modbus_var[0] :=%IW0;
Temp_chilled_medium_out:=wordstoReal(modbus_var_1000[0],modbus_var_1000[1]);
Temp_chilled_medium_in:=wordstoReal(modbus_var_1000[2],modbus_var_1000[3]);
Temp_water_inlet_cond:=wordstoReal(modbus_var_1000[4],modbus_var_1000[5]);
Temp_water_outlet_cond:=wordstoReal(modbus_var_1000[6],modbus_var_1000[7]);
SP_CW_controller:=wordstoReal(modbus_var_1000[8],modbus_var_1000[9]);
SP_PID_seawater:=wordstoReal(modbus_var_1000[10],modbus_var_1000[11]);
COP_chiller_mech:=wordstoReal(modbus_var_1000[12],modbus_var_1000[13]);
P2_mot_1_kW:=wordstoReal(modbus_var_1000[14],modbus_var_1000[15]);
Thrust_bearing_ref:=wordstoReal(modbus_var_1000[16],modbus_var_1000[17]);
Thrust_bearing_ref_min:=wordstoReal(modbus_var_1000[18],modbus_var_1000[19]);
Thrust_bearing_ref_max:=wordstoReal(modbus_var_1000[20],modbus_var_1000[21]);
Press_suction_compr:=wordstoReal(modbus_var_1000[22],modbus_var_1000[23]);
Press_discharge_compr:=wordstoReal(modbus_var_1000[24],modbus_var_1000[25]);
Suction_saturated_temp:=wordstoReal(modbus_var_1000[26],modbus_var_1000[27]);
Discharge_saturated_temp:=wordstoReal(modbus_var_1000[28],modbus_var_1000[29]);
Temp_discharge:=wordstoReal(modbus_var_1000[30],modbus_var_1000[31]);
Discharge_superheat:=wordstoReal(modbus_var_1000[32],modbus_var_1000[33]);
Liquid_level_condenser:=wordstoReal(modbus_var_1000[34],modbus_var_1000[35]);
Feedback_liquid_valve:=wordstoReal(modbus_var_1000[36],modbus_var_1000[37]);
Feedback_HGV:=wordstoReal(modbus_var_1000[38],modbus_var_1000[39]);
Spare_0:=wordstoReal(modbus_var_1000[40],modbus_var_1000[41]);
Chiller_capacity_kW:=wordstoReal(modbus_var_1000[42],modbus_var_1000[43]);
Motor_current:=wordstoReal(modbus_var_1000[44],modbus_var_1000[45]);
SP_MC_controller:=wordstoReal(modbus_var_1000[46],modbus_var_1000[47]);
Running_hours_compressormotor:=wordstoReal(modbus_var_1000[48],modbus_var_1000[49]);   //wordstoReal yes
//Running_hours_compressormotor:=wordstoDword(modbus_var_1000[48],modbus_var_1000[49]);     //wordstoDword nope
Chiller_capacity_t1:=wordstoReal(modbus_var_1000[50],modbus_var_1000[51]);
Thrust_bearing_position:=wordstoReal(modbus_var_1000[52],modbus_var_1000[53]);
Feedback_PRV:=wordstoReal(modbus_var_1000[54],modbus_var_1000[55]);
Prerotary_output:=wordstoReal(modbus_var_1000[56],modbus_var_1000[57]);
Feedback_VGD:=wordstoReal(modbus_var_1000[58],modbus_var_1000[59]);
VGD_output:=wordstoReal(modbus_var_1000[60],modbus_var_1000[61]);
Hot_gas_valve_output:=wordstoReal(modbus_var_1000[62],modbus_var_1000[63]);
Anti_recycle_time:=wordstoReal(modbus_var_1000[64],modbus_var_1000[65]);
Spare:=wordstoReal(modbus_var_1000[66],modbus_var_1000[67]);
Speed_feedback_VFD:=wordstoReal(modbus_var_1000[68],modbus_var_1000[69]);
Spare:=wordstoReal(modbus_var_1000[70],modbus_var_1000[71]);
Stall_detector:=wordstoReal(modbus_var_1000[72],modbus_var_1000[73]);
Chiller_capacity:=wordstoReal(modbus_var_1000[74],modbus_var_1000[75]);
Spare:=wordstoReal(modbus_var_1000[76],modbus_var_1000[77]);
Spare:=wordstoReal(modbus_var_1000[78],modbus_var_1000[79]);
Press_oil_receiver:=wordstoReal(modbus_var_1000[80],modbus_var_1000[81]);
Press_oil_compr:=wordstoReal(modbus_var_1000[82],modbus_var_1000[83]);
Oil_pressure_before_filter:=wordstoReal(modbus_var_1000[84],modbus_var_1000[85]);
Oil_diff_pressure:=wordstoReal(modbus_var_1000[86],modbus_var_1000[87]);
SP_freq_oil_pump_VFD:=wordstoReal(modbus_var_1000[88],modbus_var_1000[89]); 
//Setpoint_conv_oil_pump:=wordstoReal(modbus_var_1000[88],modbus_var_1000[89]); 
Oil_temp_receiver:=wordstoReal(modbus_var_1000[90],modbus_var_1000[91]);
Temp_oil_inlet_compr:=wordstoReal(modbus_var_1000[92],modbus_var_1000[93]);
SP_oil_pressure_diff:=wordstoReal(modbus_var_1000[94],modbus_var_1000[95]);
Oil_pump_running_hours:=wordstoReal(modbus_var_1000[96],modbus_var_1000[97]);
Spare:=wordstoReal(modbus_var_1000[98],modbus_var_1000[99]);
Spare:=wordstoReal(modbus_var_1000[100],modbus_var_1000[101]);
Spare:=wordstoReal(modbus_var_1000[102],modbus_var_1000[103]);
Press_chilled_medium_out:=wordstoReal(modbus_var_1000[104],modbus_var_1000[105]);
Press_chilled_medium_in:=wordstoReal(modbus_var_1000[106],modbus_var_1000[107]);
Press_water_cond_out:=wordstoReal(modbus_var_1000[108],modbus_var_1000[109]);
Press_water_cond_inlet:=wordstoReal(modbus_var_1000[110],modbus_var_1000[111]);
dP_CW:=wordstoReal(modbus_var_1000[112],modbus_var_1000[113]);
dP_SW:=wordstoReal(modbus_var_1000[114],modbus_var_1000[115]);
Feedback_seawater_valve_overboard:=wordstoReal(modbus_var_1000[116],modbus_var_1000[117]);
Spare:=wordstoReal(modbus_var_1000[118],modbus_var_1000[119]);
Spare:=wordstoReal(modbus_var_1000[120],modbus_var_1000[121]);
Spare:=wordstoReal(modbus_var_1000[122],modbus_var_1000[123]);
Temp_motor_wind_R:=wordstoReal(modbus_var_1001[124],modbus_var_1001[125]);
Temp_motor_wind_S:=wordstoReal(modbus_var_1001[126],modbus_var_1001[127]);
Temp_motor_wind_T:=wordstoReal(modbus_var_1001[128],modbus_var_1001[129]);
Max_motor_wind_temp:=wordstoReal(modbus_var_1001[130],modbus_var_1001[131]);
Temp_motor_air:=wordstoReal(modbus_var_1001[132],modbus_var_1001[133]);
Temp_motor_bearing_DE:=wordstoReal(modbus_var_1001[134],modbus_var_1001[135]);
Temp_motor_bearing_NDE:=wordstoReal(modbus_var_1001[136],modbus_var_1001[137]);
Vibration_compressor_DE:=wordstoReal(modbus_var_1001[138],modbus_var_1001[139]);
Vibration_compressor_NDE:=wordstoReal(modbus_var_1001[140],modbus_var_1001[141]);
SW_pump_speed_order:=wordstoReal(modbus_var_1001[142],modbus_var_1001[143]);
Order_SWW_overboard:=wordstoReal(modbus_var_1001[144],modbus_var_1001[145]);
Control_signal_SW_valve:=wordstoReal(modbus_var_1001[144],modbus_var_1001[145]);   
Order_SWW_bypass:=wordstoReal(modbus_var_1001[146],modbus_var_1001[147]);
Liquid_valve_output:=wordstoReal(modbus_var_1001[148],modbus_var_1001[149]);
SP_cond_press:=wordstoReal(modbus_var_1001[150],modbus_var_1001[151]);
SP_PID_Level:=wordstoReal(modbus_var_1001[152],modbus_var_1001[153]);  //mer rätt AO?
//SP_t1:=wordstoReal(modbus_var_1001[152],modbus_var_1001[153]);       // vad är detta måste kollas  SP Condenser level? PT   Tror Discharge pressure setpoint AÖ
Oil_Filter_Drop:=wordstoReal(modbus_var_1001[154],modbus_var_1001[155]);    
Min_allowed_PRVposition:=wordstoReal(modbus_var_1001[156],modbus_var_1001[157]); 
Stall_ramp:=wordstoReal(modbus_var_1001[158],modbus_var_1001[159]);
Theta_out:=wordstoReal(modbus_var_1001[160],modbus_var_1001[161]);
Control_signal_unit_d:=wordstoReal(modbus_var_1001[162],modbus_var_1001[163]);    // Sequence control signal  PT
Order_VFD_perc:=wordstoReal(modbus_var_1001[164],modbus_var_1001[165]); 
Order_VFD_Hz:=wordstoReal(modbus_var_1001[166],modbus_var_1001[167]);
Speed_feedback_VFD:=wordstoReal(modbus_var_1001[168],modbus_var_1001[169]);
Opt_speed_VFD_perc:=wordstoReal(modbus_var_1001[170],modbus_var_1001[171]);
Opt_speed_VFD_Hz:=wordstoReal(modbus_var_1001[172],modbus_var_1001[173]);
Spare:=wordstoReal(modbus_var_1001[174],modbus_var_1001[175]);
P1_motor_kW:=wordstoReal(modbus_var_1001[176],modbus_var_1001[177]);
COP_chiller_ele:=wordstoReal(modbus_var_1001[178],modbus_var_1001[179]);
PI_chiller:=wordstoReal(modbus_var_1001[180],modbus_var_1001[181]);
Wasted_energy_kW:=wordstoReal(modbus_var_1001[182],modbus_var_1001[183]);
Cal_date_MMYY:=wordstoReal(modbus_var_1001[184],modbus_var_1001[185]);
Spare:=wordstoReal(modbus_var_1001[186],modbus_var_1001[187]);
Spare:=wordstoReal(modbus_var_1001[188],modbus_var_1001[189]);
Spare:=wordstoReal(modbus_var_1001[190],modbus_var_1001[191]);
Spare:=wordstoReal(modbus_var_1001[192],modbus_var_1001[193]);
Spare:=wordstoReal(modbus_var_1001[194],modbus_var_1001[195]);
Spare:=wordstoReal(modbus_var_1001[196],modbus_var_1001[197]);
Spare:=wordstoReal(modbus_var_1001[198],modbus_var_1001[199]);
Spare:=wordstoReal(modbus_var_1001[200],modbus_var_1001[201]);
Spare:=wordstoReal(modbus_var_1001[202],modbus_var_1001[203]);
Spare:=wordstoReal(modbus_var_1001[204],modbus_var_1001[205]);
Spare:=wordstoReal(modbus_var_1001[206],modbus_var_1001[207]);
Spare:=wordstoReal(modbus_var_1001[208],modbus_var_1001[209]);
Spare:=wordstoReal(modbus_var_1001[210],modbus_var_1001[211]);

// Write PI to PLC
modbus_var_1001[180]:=modbusslave_com.sequence_highByte_PI_ch_1;
modbus_var_1001[181]:=modbusslave_com.sequence_lowByte_PI_ch_1;
modbus_var_1001[182]:=modbusslave_com.sequence_highByte_Wasted_energy_ch_1_kW;
modbus_var_1001[183]:=modbusslave_com.sequence_lowByte_Wasted_energy_ch_1_kW;

// Word variables
Alarm_limit_stall_count_unscaled:=modbus_var_1001[211];
Alarm_limit_stall_count:=Alarm_limit_stall_count_unscaled*1.0;
Sec_above_stall_limit:=scaleFunction(modbus_var_1001[212],1.0, 0);
Min_above_stall_limit:=scaleFunction(modbus_var_1001[213],1.0, 0);
Hrs_above_stall_limit:=scaleFunction(modbus_var_1001[214],1.0, 0);
Days_above_stall_limit:=scaleFunction(modbus_var_1001[215],1.0, 0);
Number_of_starts:=scaleFunction(modbus_var_1001[216],1.0, 0);
Q2_chillerMWh:=scaleFunction(modbus_var_1001[217],1.0, 0); 
Chiller_P2_MWh:=scaleFunction(modbus_var_1001[218],1.0, 0);
Surge_counter_VFD:=scaleFunction(modbus_var_1001[219],1.0, 0);

Trip_BITs_0_to_15:=modbus_var_1002[320];
Trip_BITs_16_to_31:=modbus_var_1002[321];
Trip_BITs_32_to_47:=modbus_var_1002[322];
Trip_BITs_48_to_63:=modbus_var_1002[323];
Trip_BITs_64_to_79:=modbus_var_1002[324];
Trip_BITs_80_to_95:=modbus_var_1002[325];
Trip_BITs_96_to_121:=modbus_var_1002[326];
Trip_BITs_122_to_137:=modbus_var_1002[327];
Trip_BITs_138_to_153:=modbus_var_1002[328];

Alarm_BITs_0_to_15:=modbus_var_1002[330];
Alarm_BITs_16_to_31:=modbus_var_1002[331];
Alarm_BITs_32_to_47:=modbus_var_1002[332];
Alarm_BITs_48_to_63:=modbus_var_1002[332];
Alarm_BITs_64_to_79:=modbus_var_1002[333];

Statusbits_0_to_15:=modbus_var_1002[300];
Statusbits_16_to_31:=modbus_var_1002[301];
Statusbits_32_to_47:=modbus_var_1002[302];
Statusbits_48_to_63:=modbus_var_1002[303];
Statusbits_64_to_79:=modbus_var_1002[304];
Statusbits_80_to_95:=modbus_var_1002[305];
Statusbits_96_to_111:=modbus_var_1002[310];
Statusbits_112_to_127:=modbus_var_1002[311];


//320
T_Overload_compressor_motor:=maskbitFunction(Trip_BITs_0_to_15,0);
T_Starter_failure_trip:=maskbitFunction(Trip_BITs_0_to_15,1);
T_Oil_pump_running_failure:=maskbitFunction(Trip_BITs_0_to_15,2);
T_Overload_oil_pump_motor:=maskbitFunction(Trip_BITs_0_to_15,3);
T_Compressor_running_failure:=maskbitFunction(Trip_BITs_0_to_15,4);
T_Softstarter_failure:=maskbitFunction(Trip_BITs_0_to_15,5);
T_Motorstarter_failure:=maskbitFunction(Trip_BITs_0_to_15,6);
T_Comp_motor_power_loss:=maskbitFunction(Trip_BITs_0_to_15,7);
T_Emergency_stop:=maskbitFunction(Trip_BITs_0_to_15,8);
T_Flow_switch_FT01:=maskbitFunction(Trip_BITs_0_to_15,9);
T_Chilled_pump_run_failure:=maskbitFunction(Trip_BITs_0_to_15,10);
T_CW_valveopen_failure:=maskbitFunction(Trip_BITs_0_to_15,11);
T_Sea_water_pump_run_failure:=maskbitFunction(Trip_BITs_0_to_15,12);
T_SW_valveopen_failure:=maskbitFunction(Trip_BITs_0_to_15,13);
T_Comp_motor_leak_detection:=maskbitFunction(Trip_BITs_0_to_15,14);
T_Cathodic_protect_sys_alarm:=maskbitFunction(Trip_BITs_0_to_15,15);
//321
T_High_discharge_pressure:=maskbitFunction(Trip_BITs_16_to_31,0);
T_Low_discharge_pressure:=maskbitFunction(Trip_BITs_16_to_31,1);
T_Low_suction_pressure:=maskbitFunction(Trip_BITs_16_to_31,2);
T_High_suction_pressure:=maskbitFunction(Trip_BITs_16_to_31,3);
T_High_discharge_temp:=maskbitFunction(Trip_BITs_16_to_31,4);
T_High_temp_oil_inlet_comp:=maskbitFunction(Trip_BITs_16_to_31,5);
T_High_temp_oil_receiver:=maskbitFunction(Trip_BITs_16_to_31,6);
T_Low_temp_oil_receiver:=maskbitFunction(Trip_BITs_16_to_31,7);
T_Low_oil_diff_pressure:=maskbitFunction(Trip_BITs_16_to_31,8);
T_High_diff_oil_pressure:=maskbitFunction(Trip_BITs_16_to_31,9);
T_High_oil_filter_diff_press:=maskbitFunction(Trip_BITs_16_to_31,10);
T_High_disch_superheat:=maskbitFunction(Trip_BITs_16_to_31,11);
T_Low_disch_superheat:=maskbitFunction(Trip_BITs_16_to_31,12);
T_Low_CW_inlet_temp:=maskbitFunction(Trip_BITs_16_to_31,13);
T_High_CW_inlet_temp:=maskbitFunction(Trip_BITs_16_to_31,14);
T_Low_CW_outlet_temp:=maskbitFunction(Trip_BITs_16_to_31,15);
//322
T_High_CW_outlet_temp:=maskbitFunction(Trip_BITs_32_to_47,0);
T_Low_chilled_medium_flow:=maskbitFunction(Trip_BITs_32_to_47,1);
T_High_chilled_medium_flow:=maskbitFunction(Trip_BITs_32_to_47,2);
T_Low_SW_inlet_temp:=maskbitFunction(Trip_BITs_32_to_47,3);
T_High_SW_inlet_temp:=maskbitFunction(Trip_BITs_32_to_47,4);
T_Low_SW_outlet_temp:=maskbitFunction(Trip_BITs_32_to_47,5);
T_High_SW_outlet_temp:=maskbitFunction(Trip_BITs_32_to_47,6);
T_Low_condenser_flow:=maskbitFunction(Trip_BITs_32_to_47,7);
T_High_condenser_flow:=maskbitFunction(Trip_BITs_32_to_47,8);
T_High_motor_wind_temp_R:=maskbitFunction(Trip_BITs_32_to_47,9);
T_High_motor_wind_temp_S:=maskbitFunction(Trip_BITs_32_to_47,10);
T_High_motor_wind_temp_T:=maskbitFunction(Trip_BITs_32_to_47,11);
T_High_comp_mot_DE_bear_temp:=maskbitFunction(Trip_BITs_32_to_47,12);
T_High_comp_mot_NDE_bear_temp:=maskbitFunction(Trip_BITs_32_to_47,13);
T_High_motor_air_temp:=maskbitFunction(Trip_BITs_32_to_47,14);
T_High_comp_mot_DE_bear_vib:=maskbitFunction(Trip_BITs_32_to_47,15);
//323
T_High_comp_mot_NDE_bear_vib:=maskbitFunction(Trip_BITs_48_to_63,0);
T_High_press_ratio:=maskbitFunction(Trip_BITs_48_to_63,1);
T_Low_press_ratio:=maskbitFunction(Trip_BITs_48_to_63,2);
T_High_CW_dP:=maskbitFunction(Trip_BITs_48_to_63,3);
T_Low_CW_dP:=maskbitFunction(Trip_BITs_48_to_63,4);
T_High_SW_dP:=maskbitFunction(Trip_BITs_48_to_63,5);
T_Low_SW_dP:=maskbitFunction(Trip_BITs_48_to_63,6);
T_Long_time_PRV:=maskbitFunction(Trip_BITs_48_to_63,7);
T_Surge_detection:=maskbitFunction(Trip_BITs_48_to_63,8);
T_Comp_thrust_bearing_position:=maskbitFunction(Trip_BITs_48_to_63,9);
T_Comp_thrust_neg_move:=maskbitFunction(Trip_BITs_48_to_63,10);
T_Comp_thrust_pos_move:=maskbitFunction(Trip_BITs_48_to_63,11);
T_VGD_fault:=maskbitFunction(Trip_BITs_48_to_63,12);
T_Low_liquid_level:=maskbitFunction(Trip_BITs_48_to_63,13);
T_Low_oilpress_prelube:=maskbitFunction(Trip_BITs_48_to_63,14);
T_Low_oilpress_standby:=maskbitFunction(Trip_BITs_48_to_63,15);
//324
T_Sensor_low_signal_AI_64 :=maskbitFunction(Trip_BITs_64_to_79,0);
T_Sensor_high_signal_AI_64 :=maskbitFunction(Trip_BITs_64_to_79,1);
T_Sensor_low_signal_AI_66 :=maskbitFunction(Trip_BITs_64_to_79,2);
T_Sensor_high_signal_AI_66 :=maskbitFunction(Trip_BITs_64_to_79,3);
T_Sensor_low_signal_AI_128 :=maskbitFunction(Trip_BITs_64_to_79,4);
T_Sensor_high_signal_AI_128 :=maskbitFunction(Trip_BITs_64_to_79,5);
T_Sensor_low_signal_AI_130 :=maskbitFunction(Trip_BITs_64_to_79,6);
T_Sensor_high_signal_AI_130 :=maskbitFunction(Trip_BITs_64_to_79,7);
T_Sensor_low_signal_AI_132 :=maskbitFunction(Trip_BITs_64_to_79,8);
T_Sensor_high_signal_AI_132 :=maskbitFunction(Trip_BITs_64_to_79,9);
T_Sensor_low_signal_AI_134 :=maskbitFunction(Trip_BITs_64_to_79,10);
T_Sensor_high_signal_AI_134 :=maskbitFunction(Trip_BITs_64_to_79,11);
T_Sensor_low_signal_AI_136 :=maskbitFunction(Trip_BITs_64_to_79,12);
T_Sensor_high_signal_AI_136 :=maskbitFunction(Trip_BITs_64_to_79,13);
T_Sensor_low_signal_AI_138 :=maskbitFunction(Trip_BITs_64_to_79,14);
T_Sensor_high_signal_AI_138 :=maskbitFunction(Trip_BITs_64_to_79,15);

T_Sensor_low_signal_AI_140 :=maskbitFunction(Trip_BITs_80_to_95,0);
T_Sensor_high_signal_AI_140 :=maskbitFunction(Trip_BITs_80_to_95,1);
T_Sensor_low_signal_AI_142 :=maskbitFunction(Trip_BITs_80_to_95,2);
T_Sensor_high_signal_AI_142 :=maskbitFunction(Trip_BITs_80_to_95,3);
T_Sensor_low_signal_AI_144 :=maskbitFunction(Trip_BITs_80_to_95,4);
T_Sensor_high_signal_AI_144 :=maskbitFunction(Trip_BITs_80_to_95,5);
T_Sensor_low_signal_AI_146 :=maskbitFunction(Trip_BITs_80_to_95,6);
T_Sensor_high_signal_AI_146 :=maskbitFunction(Trip_BITs_80_to_95,7);
T_Sensor_low_signal_AI_148 :=maskbitFunction(Trip_BITs_80_to_95,8);
T_Sensor_high_signal_AI_148 :=maskbitFunction(Trip_BITs_80_to_95,9);
T_Sensor_low_signal_AI_150 :=maskbitFunction(Trip_BITs_80_to_95,10);
T_Sensor_high_signal_AI_150 :=maskbitFunction(Trip_BITs_80_to_95,11);
T_Sensor_low_signal_AI_152 :=maskbitFunction(Trip_BITs_80_to_95,12);
T_Sensor_high_signal_AI_152 :=maskbitFunction(Trip_BITs_80_to_95,13);
T_Sensor_low_signal_AI_154 :=maskbitFunction(Trip_BITs_80_to_95,14);
T_Sensor_high_signal_AI_154 :=maskbitFunction(Trip_BITs_80_to_95,15);

T_Sensor_low_signal_AI_156 :=maskbitFunction(Trip_BITs_96_to_121,0);
T_Sensor_high_signal_AI_156 :=maskbitFunction(Trip_BITs_96_to_121,1);
T_Sensor_low_signal_AI_158 :=maskbitFunction(Trip_BITs_96_to_121,2);
T_Sensor_high_signal_AI_158 :=maskbitFunction(Trip_BITs_96_to_121,3);
T_Sensor_low_signal_AI_160 :=maskbitFunction(Trip_BITs_96_to_121,4);
T_Sensor_high_signal_AI_160 :=maskbitFunction(Trip_BITs_96_to_121,5);
T_Sensor_low_signal_AI_162 :=maskbitFunction(Trip_BITs_96_to_121,6);
T_Sensor_high_signal_AI_162 :=maskbitFunction(Trip_BITs_96_to_121,7);
T_Sensor_low_signal_AI_164 :=maskbitFunction(Trip_BITs_96_to_121,8);
T_Sensor_high_signal_AI_164 :=maskbitFunction(Trip_BITs_96_to_121,9);
T_Sensor_low_signal_AI_166 :=maskbitFunction(Trip_BITs_96_to_121,10);
T_Sensor_high_signal_AI_166 :=maskbitFunction(Trip_BITs_96_to_121,11);
T_Sensor_low_signal_AI_168 :=maskbitFunction(Trip_BITs_96_to_121,12);
T_Sensor_high_signal_AI_168 :=maskbitFunction(Trip_BITs_96_to_121,13);
T_Sensor_low_signal_AI_170 :=maskbitFunction(Trip_BITs_96_to_121,14);
T_Sensor_high_signal_AI_170 :=maskbitFunction(Trip_BITs_96_to_121,15);

T_Sensor_low_signal_AI_172 :=maskbitFunction(Trip_BITs_122_to_137,0);
T_Sensor_high_signal_AI_172 :=maskbitFunction(Trip_BITs_122_to_137,1);
T_Sensor_low_signal_AI_174 :=maskbitFunction(Trip_BITs_122_to_137,2);
T_Sensor_high_signal_AI_174 :=maskbitFunction(Trip_BITs_122_to_137,3);
T_Sensor_high_signal_AI_176 :=maskbitFunction(Trip_BITs_122_to_137,4);
T_Sensor_high_signal_AI_178 :=maskbitFunction(Trip_BITs_122_to_137,5);
T_Sensor_high_signal_AI_180 :=maskbitFunction(Trip_BITs_122_to_137,6);
T_Sensor_high_signal_AI_182 :=maskbitFunction(Trip_BITs_122_to_137,7);
T_Sensor_high_signal_AI_184 :=maskbitFunction(Trip_BITs_122_to_137,8);
T_Sensor_high_signal_AI_186 :=maskbitFunction(Trip_BITs_122_to_137,9);
T_Sensor_high_signal_AI_188 :=maskbitFunction(Trip_BITs_122_to_137,10);
T_Sensor_high_signal_AI_190 :=maskbitFunction(Trip_BITs_122_to_137,11);
T_Sensor_high_signal_AI_192 :=maskbitFunction(Trip_BITs_122_to_137,12);
T_Sensor_high_signal_AI_194 :=maskbitFunction(Trip_BITs_122_to_137,13);
T_Sensor_high_signal_AI_196 :=maskbitFunction(Trip_BITs_122_to_137,14);
T_Sensor_high_signal_AI_198 :=maskbitFunction(Trip_BITs_122_to_137,15);

T_Sensor_high_signal_AI_200 :=maskbitFunction(Trip_BITs_138_to_153,0);
T_Sensor_high_signal_AI_202 :=maskbitFunction(Trip_BITs_138_to_153,1);
T_Sensor_high_signal_AI_204 :=maskbitFunction(Trip_BITs_138_to_153,2);
T_Sensor_high_signal_AI_206:=maskbitFunction(Trip_BITs_138_to_153,3);

// Alarm bits 330
A_High_control_panel_temp:=maskbitFunction(Alarm_BITs_0_to_15,0);
A_high_disch_press:=maskbitFunction(Alarm_BITs_0_to_15,1);
A_low_disch_press :=maskbitFunction(Alarm_BITs_0_to_15,2);
A_Low_suction_pressure:=maskbitFunction(Alarm_BITs_0_to_15,3);
A_High_suction_pressure:=maskbitFunction(Alarm_BITs_0_to_15,4);
A_High_discharge_temp :=maskbitFunction(Alarm_BITs_0_to_15,5);
A_High_temp_oil_inlet_comp:=maskbitFunction(Alarm_BITs_0_to_15,6);
A_Low_temp_oil_inlet_comp:=maskbitFunction(Alarm_BITs_0_to_15,7);
A_High_oil_temp_receiver:=maskbitFunction(Alarm_BITs_0_to_15,8);
A_Low_oil_temp_receiver:=maskbitFunction(Alarm_BITs_0_to_15,9);
A_Low_oil_diff_pressure:=maskbitFunction(Alarm_BITs_0_to_15,10);
A_High_oil_diff_pressure:=maskbitFunction(Alarm_BITs_0_to_15,11);
A_High_discharge_superheat:=maskbitFunction(Alarm_BITs_0_to_15,12);
A_Low_discharge_superheat:=maskbitFunction(Alarm_BITs_0_to_15,13);
A_Low_CW_inlet_temp:=maskbitFunction(Alarm_BITs_0_to_15,14);
A_High_CW_inlet_temp:=maskbitFunction(Alarm_BITs_0_to_15,15);
//331
A_Low_CW_outlet_temp:=maskbitFunction(Alarm_BITs_16_to_31,0);
A_High_CW_outlet_temp:=maskbitFunction(Alarm_BITs_16_to_31,1);
A_Low_chilled_medium_flow:=maskbitFunction(Alarm_BITs_16_to_31,2);
A_High_chilled_medium_flow:=maskbitFunction(Alarm_BITs_16_to_31,3);
A_Low_condenser_flow:=maskbitFunction(Alarm_BITs_16_to_31,4);
A_High_condenser_flow:=maskbitFunction(Alarm_BITs_16_to_31,5);
A_High_press_ratio:=maskbitFunction(Alarm_BITs_16_to_31,6);
A_Low_press_ratio:=maskbitFunction(Alarm_BITs_16_to_31,7);
A_Motor_speed_low :=maskbitFunction(Alarm_BITs_16_to_31,8);
A_Low_SW_inlet_temp:=maskbitFunction(Alarm_BITs_16_to_31,9); 
A_High_SW_inlet_temp:=maskbitFunction(Alarm_BITs_16_to_31,10); 
A_Low_SW_outlet_temp:=maskbitFunction(Alarm_BITs_16_to_31,11); 
A_High_SW_outlet_temp:=maskbitFunction(Alarm_BITs_16_to_31,12);
A_High_suction_superheat:=maskbitFunction(Alarm_BITs_16_to_31,13);
A_Low_suction_superheat:=maskbitFunction(Alarm_BITs_16_to_31,14);
A_High_oil_filter_diff_press:=maskbitFunction(Alarm_BITs_16_to_31,15);
//332
A_High_CW_dP:=maskbitFunction(Alarm_BITs_32_to_47,0);
A_Low_CW_dP:=maskbitFunction(Alarm_BITs_32_to_47,1);
A_High_temp_oil_separator:=maskbitFunction(Alarm_BITs_32_to_47,2);
A_Low_temp_oil_separator:=maskbitFunction(Alarm_BITs_32_to_47,3);
A_High_motor_wind_temp_R:=maskbitFunction(Alarm_BITs_32_to_47,4);
A_High_motor_wind_temp_S:=maskbitFunction(Alarm_BITs_32_to_47,5);
A_High_motor_wind_temp_T:=maskbitFunction(Alarm_BITs_32_to_47,6);
A_High_comp_mo_DE_bear_temp:=maskbitFunction(Alarm_BITs_32_to_47,7);
A_High_comp_mo_NDE_bear_temp:=maskbitFunction(Alarm_BITs_32_to_47,8);
A_High_motor_air_temp:=maskbitFunction(Alarm_BITs_32_to_47,9);
A_High_comp_mo_DE_bear_vib:=maskbitFunction(Alarm_BITs_32_to_47,10);
A_High_comp_mo_NDE_bear_vib:=maskbitFunction(Alarm_BITs_32_to_47,11);
//A_High_CW_dP:=maskbitFunction(Alarm_BITs_32_to_47,12);                       //Double defined?
//A_Low_CW_dP:=maskbitFunction(Alarm_BITs_32_to_47,13);                        //Double defined?
A_High_SW_dP:=maskbitFunction(Alarm_BITs_32_to_47,14);                       
A_Low_SW_dP:=maskbitFunction(Alarm_BITs_32_to_47,15);
//333
A_VGD_fault:=maskbitFunction(Alarm_BITs_48_to_63,0);
//A_Rotating_stall:=maskbitFunction(Alarm_BITs_48_to_63,0);  // kollas
A_Low_liquid_level:=maskbitFunction(Alarm_BITs_48_to_63,1);





// Statusbits 310
Unit_running:=maskbitFunction(Statusbits_96_to_111,0);
Unit_trip:=maskbitFunction(Statusbits_96_to_111,1);
Unit_alarm:=maskbitFunction(Statusbits_96_to_111,2);
Unit_remote:=maskbitFunction(Statusbits_96_to_111,3);
Unit_auto:=maskbitFunction(Statusbits_96_to_111,4);
Unit_manual:=maskbitFunction(Statusbits_96_to_111,5);
Unit_available:=maskbitFunction(Statusbits_96_to_111,6);
Unit_start_switch:=maskbitFunction(Statusbits_96_to_111,7);
Comp_oil_pump:=maskbitFunction(Statusbits_96_to_111,8);
Oil_heater:=maskbitFunction(Statusbits_96_to_111,9);
Solenoid_oil_return:=maskbitFunction(Statusbits_96_to_111,10);
Solenoid_liquid_inj:=maskbitFunction(Statusbits_96_to_111,11);
Low_oil_temperature:=maskbitFunction(Statusbits_96_to_111,12);
Sea_water_pump:=maskbitFunction(Statusbits_96_to_111,13);
CW_Flow_ind:=maskbitFunction(Statusbits_96_to_111,14);
Start_inhib_time_between_start:=maskbitFunction(Statusbits_96_to_111,15);
// Statusbits 311
Start_inhib_time_beetween_stop:=maskbitFunction(Statusbits_112_to_127,0);
Start_inhib_PRV_not_min:=maskbitFunction(Statusbits_112_to_127,1);
Start_inhib_Motor_overload:=maskbitFunction(Statusbits_112_to_127,2);
VFD_ready:=maskbitFunction(Statusbits_112_to_127,3);
VFD_ramp_100_perc:=maskbitFunction(Statusbits_112_to_127,4);
VFD_locked_100_perc:=maskbitFunction(Statusbits_112_to_127,5);
VFD_ramp_d_PRVcontrol:=maskbitFunction(Statusbits_112_to_127,6);
PRV_control:=maskbitFunction(Statusbits_112_to_127,7);
VFD_control:=maskbitFunction(Statusbits_112_to_127,8);
S_Spare_1:=maskbitFunction(Statusbits_112_to_127,9);
S_Spare_1:=maskbitFunction(Statusbits_112_to_127,10);
S_Spare_1:=maskbitFunction(Statusbits_112_to_127,11);
S_Spare_1:=maskbitFunction(Statusbits_112_to_127,12);
S_Spare_1:=maskbitFunction(Statusbits_112_to_127,13);
S_Spare_1:=maskbitFunction(Statusbits_112_to_127,14);
S_Spare_1:=maskbitFunction(Statusbits_112_to_127,15);

DI_0_0:=maskbitFunction(Statusbits_0_to_15,0);
DI_0_1:=maskbitFunction(Statusbits_0_to_15,1);
DI_0_2:=maskbitFunction(Statusbits_0_to_15,2);
DI_0_3:=maskbitFunction(Statusbits_0_to_15,3);
DI_0_4:=maskbitFunction(Statusbits_0_to_15,4);
DI_0_5:=maskbitFunction(Statusbits_0_to_15,5);
DI_0_6:=maskbitFunction(Statusbits_0_to_15,6);
DI_0_7:=maskbitFunction(Statusbits_0_to_15,7);
DI_1_0:=maskbitFunction(Statusbits_0_to_15,8);
DI_1_1:=maskbitFunction(Statusbits_0_to_15,9);
DI_1_2:=maskbitFunction(Statusbits_0_to_15,10);
DI_1_3:=maskbitFunction(Statusbits_0_to_15,11);
DI_1_4:=maskbitFunction(Statusbits_0_to_15,12);
DI_1_5:=maskbitFunction(Statusbits_0_to_15,13);
DI_8_0:=maskbitFunction(Statusbits_0_to_15,14);
DI_8_1:=maskbitFunction(Statusbits_0_to_15,15);

DI_8_2:=maskbitFunction(Statusbits_16_to_31,0);
DI_8_3:=maskbitFunction(Statusbits_16_to_31,1);
DI_8_4:=maskbitFunction(Statusbits_16_to_31,2);
DI_8_5:=maskbitFunction(Statusbits_16_to_31,3);
DI_8_6:=maskbitFunction(Statusbits_16_to_31,4);
DI_8_7:=maskbitFunction(Statusbits_16_to_31,5);
DI_9_0:=maskbitFunction(Statusbits_16_to_31,6);
DI_9_1:=maskbitFunction(Statusbits_16_to_31,7);
DI_9_2:=maskbitFunction(Statusbits_16_to_31,8);
DI_9_3:=maskbitFunction(Statusbits_16_to_31,9);
DI_9_4:=maskbitFunction(Statusbits_16_to_31,10);
DI_9_5:=maskbitFunction(Statusbits_16_to_31,11);
DI_9_6:=maskbitFunction(Statusbits_16_to_31,12);
DI_9_7:=maskbitFunction(Statusbits_16_to_31,13);
T_Spare_3:=maskbitFunction(Statusbits_16_to_31,14);
T_Spare_3:=maskbitFunction(Statusbits_16_to_31,15);

DO_0_0:=maskbitFunction(Statusbits_32_to_47,0);
DO_0_1:=maskbitFunction(Statusbits_32_to_47,1);
DO_0_2:=maskbitFunction(Statusbits_32_to_47,2);
DO_0_3:=maskbitFunction(Statusbits_32_to_47,3);
DO_0_4:=maskbitFunction(Statusbits_32_to_47,4);
DO_0_5:=maskbitFunction(Statusbits_32_to_47,5);
DO_0_6:=maskbitFunction(Statusbits_32_to_47,6);
DO_0_7:=maskbitFunction(Statusbits_32_to_47,7);
DO_1_0:=maskbitFunction(Statusbits_32_to_47,8);
DO_1_1:=maskbitFunction(Statusbits_32_to_47,9);
DO_8_0:=maskbitFunction(Statusbits_32_to_47,10);
DO_8_1:=maskbitFunction(Statusbits_32_to_47,11);
DO_8_2:=maskbitFunction(Statusbits_32_to_47,12);
DO_8_3:=maskbitFunction(Statusbits_32_to_47,13);
DO_8_4:=maskbitFunction(Statusbits_32_to_47,14);
DO_8_5:=maskbitFunction(Statusbits_32_to_47,15);

DO_8_6:=maskbitFunction(Statusbits_48_to_63,0);
DO_8_7:=maskbitFunction(Statusbits_48_to_63,1);
DO_9_0:=maskbitFunction(Statusbits_48_to_63,2);
DO_9_1:=maskbitFunction(Statusbits_48_to_63,3);
DO_9_2:=maskbitFunction(Statusbits_48_to_63,4);
DO_9_3:=maskbitFunction(Statusbits_48_to_63,5);
DO_9_4:=maskbitFunction(Statusbits_48_to_63,6);
DO_9_5:=maskbitFunction(Statusbits_48_to_63,7);
DO_9_6:=maskbitFunction(Statusbits_48_to_63,8);
DO_9_7:=maskbitFunction(Statusbits_48_to_63,9);
DO_12_0:=maskbitFunction(Statusbits_48_to_63,10);
DO_12_1:=maskbitFunction(Statusbits_48_to_63,11);
DO_12_2:=maskbitFunction(Statusbits_48_to_63,12);
DO_12_3:=maskbitFunction(Statusbits_48_to_63,13);
DO_12_4:=maskbitFunction(Statusbits_48_to_63,14);
DO_12_5:=maskbitFunction(Statusbits_48_to_63,15);

DO_12_6:=maskbitFunction(Statusbits_64_to_79,0);
DO_12_7:=maskbitFunction(Statusbits_64_to_79,1);
T_Spare_3:=maskbitFunction(Statusbits_64_to_79,2);
T_Spare_3:=maskbitFunction(Statusbits_64_to_79,3);
T_Spare_3:=maskbitFunction(Statusbits_64_to_79,4);
T_Spare_3:=maskbitFunction(Statusbits_64_to_79,5);
T_Spare_3:=maskbitFunction(Statusbits_64_to_79,6);
T_Spare_3:=maskbitFunction(Statusbits_64_to_79,7);
T_Spare_3:=maskbitFunction(Statusbits_64_to_79,8);
T_Spare_3:=maskbitFunction(Statusbits_64_to_79,9);
T_Spare_3:=maskbitFunction(Statusbits_64_to_79,10);
T_Spare_3:=maskbitFunction(Statusbits_64_to_79,11);
T_Spare_3:=maskbitFunction(Statusbits_64_to_79,12);
T_Spare_3:=maskbitFunction(Statusbits_64_to_79,13);
T_Spare_3:=maskbitFunction(Statusbits_64_to_79,14);
T_Spare_3:=maskbitFunction(Statusbits_64_to_79,15);



// Graphic controls
IF Unit_remote THEN
	Unit_switch_status:=2;
ELSIF Unit_auto THEN 
	Unit_switch_status:=3;
ELSIF Unit_manual THEN 
	Unit_switch_status:=4;

END_IF ;	

IF select_trendvalue > 0 THEN
	show_trendvalue[select_trendvalue]:= TRUE;
ELSIF select_trendvalue = 0 THEN
	FOR i := 0 TO 50 DO
      show_trendvalue[i] := FALSE;
   	END_FOR
END_IF ;	
	
// timer2 (IN:= TRUE, PT:=T#5S);;
//	IF timer2_Q THEN
//		Temp_motor_bearing_DE := Temp_motor_bearing_DE +1;
//		Motor_current := Motor_current + 1 ;
//		Timer2(IN:= FALSE);
//	END_IF

END_PROGRAM

// Calculus
PROGRAM Calculus
VAR


// MWCC

NakW_chiller_3 : REAL ;
NakW_chiller_4 : REAL ;

COP_chiller_3 : REAL ;
COP_chiller_4 : REAL ;
NakW_chiller_5 : REAL ;
NakW_chiller_6 : REAL ;

COP_chiller_5 : REAL ;
COP_chiller_6 : REAL ;
{attribute 'ac_datalog_hysteresis' := '100'}
{attribute 'ac_datalog' := 'DatalogChannel'}
Tot_Power_motor : REAL ;
{attribute 'ac_datalog_hysteresis' := '300'}
{attribute 'ac_datalog' := 'DatalogChannel'}
Tot_Q2 : REAL ;
{attribute 'ac_datalog_hysteresis' := '100'}
{attribute 'ac_datalog' := 'DatalogChannel'}
Tot_Q2_MWh : REAL ;
{attribute 'ac_datalog_hysteresis' := '100'}
{attribute 'ac_datalog' := 'DatalogChannel'}
Tot_P1_MWh : REAL ;
Power_motor_3_kW : REAL ;
Power_motor_4_kW : REAL ;
Power_motor_5_kW : REAL ;
Power_motor_6_kW : REAL ;
Power_3_not_zero : REAL ;
Power_4_not_zero : REAL ;
Power_5_not_zero : REAL ;
Power_6_not_zero : REAL ;

// SE700
Q2kW_chiller_1 : REAL ;
Q2kW_chiller_2 : REAL ;
Chiller_1_dpCW_bar : REAL ;
Chiller_2_dpCW_bar : REAL ;
Chiller_1_SR_dpCW_bar : REAL ;
Chiller_2_SR_dpCW_bar : REAL ;
Power_motor_1_kW : REAL ;
Power_motor_2_kW : REAL ;
Power_1_not_zero : REAL ;
Power_2_not_zero : REAL ;
NakW_chiller_1 : REAL ;
NakW_chiller_2 : REAL ;
COP_chiller_1 : REAL ;
COP_chiller_2 : REAL ;



Power_3_not_zero_func: WORD := 100;
Power_4_not_zero_func :  WORD := 100;
COP_chiller_3_func :  WORD := 100;
COP_chiller_4_func :  WORD := 100;
Power_5_not_zero_func: WORD := 100;
Power_6_not_zero_func :  WORD := 100;
COP_chiller_5_func :  WORD := 100;
COP_chiller_6_func :  WORD := 100;
Tot_Power_motor_func :  WORD := 100;
Tot_Q2_func :  WORD := 100;
Tot_Q2_MWh_func :  WORD := 100;
Tot_Na_MWh_func :  WORD := 100;
Power_motor_3_kW_func :  WORD := 100;
Power_motor_4_kW_func :  WORD := 100;

// SE700

Man_Auto_Chiller_1_func :  WORD := 100;
Man_Auto_Chiller_2_func :  WORD := 100;
//SE700_Chiller_1_Modb|||VALISERR(LOCAL.MODBUS2.Chiller_1.Program_number);//
//SE700_Chiller_2_Modb|||VALISERR(LOCAL.MODBUS2.Chiller_2.Program_number);
Flow_factor_chiller1_func :  WORD := 100;
Flow_factor_chiller2_func :  WORD := 100;


SR_Nom_dP_bar_func :  WORD := 100;


Chiller_1_dT_func :  WORD := 100;
Chiller_2_dT_func :  WORD := 100;
Chiller_1_max_dT_func :  WORD := 100;
Chiller_2_max_dT_func :  WORD := 100;
Chiller_1_Capacity_func :  WORD := 100;
Chiller_2_Capacity_func :  WORD := 100;
Chiller_1_CapacitykW_func :  WORD := 100;
Chiller_2_CapacitykW_func :  WORD := 100;
Chiller_1_dpCW_bar_func :  WORD := 100;
Chiller_2_dpCW_bar_func :  WORD := 100;
Chiller_1_SR_dpCW_bar_func :  WORD := 100;
Chiller_2_SR_dpCW_bar_func :  WORD := 100;
Power_motor_1_kW_func :  WORD := 100;
Power_motor_2_kW_func :  WORD := 100;
Power_1_not_zero_func :  WORD := 100;
Power_2_not_zero_func :  WORD := 100;
COP_chiller_1_func :  WORD := 100;
COP_chiller_2_func :  WORD := 100;
Chiller_1_Capacity_corr_flow_factor_func :  WORD := 100;
Chiller_2_Capacity_corr_flow_factor_func :  WORD := 100;
// New Variables
PI_chiller_1  : REAL ;
PI_chiller_1_word : WORD ;
PI_Calc_Error_AC1 : BOOL ;
PI_chiller_2  : REAL ;
PI_chiller_2_word : WORD ;
PI_Calc_Error_AC2 : BOOL ;
PI_chiller_3  : REAL ;
PI_chiller_3_word : WORD ;
PI_Calc_Error_AC3 : BOOL ;
PI_chiller_4  : REAL ;
PI_chiller_4_word : WORD ;
PI_Calc_Error_AC4 : BOOL ;
PI_chiller_5  : REAL ;
PI_chiller_5_word : WORD ;
PI_Calc_Error_AC5 : BOOL ;
PI_chiller_6  : REAL ;
PI_chiller_6_word : WORD ;
PI_Calc_Error_AC6 : BOOL ;
delaytimer2 : TON ;	
resetbuttons : BOOL := FALSE  ;
COP_theo_AC1 :REAL ;	
COP_theo_AC2 :REAL ;
COP_theo_AC3 :REAL ;
COP_theo_AC4 :REAL ;
COP_theo_AC5 :REAL ;
COP_theo_AC6 :REAL ;
totRunningChillers : INT;
WastedEnergy_AC1 :REAL ;
WastedEnergy_AC1_word :WORD ;
WastedEnergy_AC2 :REAL ;
WastedEnergy_AC2_word :WORD ;
WastedEnergy_AC3 :REAL ;
WastedEnergy_AC3_word :WORD ;
WastedEnergy_AC4 :REAL ;
WastedEnergy_AC4_word :WORD ;
WastedEnergy_AC5 :REAL ;
WastedEnergy_AC5_word :WORD ;
WastedEnergy_AC6 :REAL ;
WastedEnergy_AC6_word :WORD ;
Total_PI : REAL ;
// Time variables
Result_time : SysTimeRtc.RTS_IEC_RESULT;
udiLocal_DateAndTime : UDINT;
current_date : UDINT ;

	
END_VAR

IF GVL.startUp THEN
	startupReadcsv();
	IF NOT GVL.startUp THEN	
		GVL.xReadCOP := FALSE;
		GVL.startdelaytimer :=TRUE;
	END_IF
	
END_IF

GVL.delaytimer (IN:= GVL.startdelaytimer, PT:=T#5S);
IF GVL.delaytimer.Q THEN
	GVL.xReadCOP := TRUE;
	GVL.startdelaytimer:=FALSE;
	resetbuttons := TRUE ;
END_IF
delaytimer2 (IN:= resetbuttons, PT:=T#5S);
IF delaytimer2.Q THEN
	GVL.xReadCOP := FALSE;
	GVL.initRead := FALSE;
	resetbuttons := FALSE;
END_IF

// Get system time
current_date := TO_UDINT(SysTimeRtcGet(Result_time));
Result_time := SysTimeRTCConvertUTCToLocal(current_date, udiLocal_DateAndTime);
GVL.CurrentDate := TO_DT(udiLocal_DateAndTime); // DT#2018-6-6-9:8:38

// MWCC
Tot_Q2_MWh:=Tot_Q2:=Chiller_1.Q2_chillerMWh + Chiller_2.Q2_chillerMWh + Chiller_3.Q2_chillerMWh + Chiller_4.Q2_chillerMWh (*+ Chiller_5.Q2_chillerMWh + Chiller_6.Q2_chillerMWh*) ;
//Tot_Q2_MWh:=Tot_Q2:=Sequence.Chiller_1_Q2_MWh + Sequence.Chiller_2_Q2_MWh + Sequence.Chiller_3_Q2_MWh + Sequence.Chiller_4_Q2_MWh + Sequence.Chiller_5_Q2_MWh + Sequence.Chiller_6_Q2_MWh ;
Tot_P1_MWh:=Tot_Q2:=Chiller_1.Chiller_P1_MWh + Chiller_2.Chiller_P1_MWh + Chiller_3.Chiller_P1_MWh + Chiller_4.Chiller_P1_MWh (*+ Chiller_5.Chiller_P1_MWh + Chiller_6.Chiller_P1_MWh*) ;
//Tot_P1_MWh:=Tot_Q2:=Sequence.Chiller_1_P1_MWh + Sequence.Chiller_2_P1_MWh + Sequence.Chiller_3_P1_MWh + Sequence.Chiller_4_P1_MWh + Sequence.Chiller_5_P1_MWh + Sequence.Chiller_6_P1_MWh ;

// New Func
Power_motor_1_kW:=Chiller_1.P1_motor_kW;
Power_motor_2_kW:=Chiller_2.P1_motor_kW;
Power_motor_3_kW:=Chiller_3.P1_motor_kW;
Power_motor_4_kW:=Chiller_4.P1_motor_kW;
//Power_motor_5_kW:=Chiller_5.P1_motor_kW;
//Power_motor_6_kW:=Chiller_6.P1_motor_kW;

Tot_Power_motor:=Power_motor_1_kW + Power_motor_2_kW + Power_motor_3_kW + Power_motor_4_kW (*+ Power_motor_5_kW + Power_motor_6_kW*);
//Tot_Q2:=sequence.Q2kW_chiller_1 + sequence.Q2kW_chiller_2 + Sequence.Q2kW_chiller_3 + Sequence.Q2kW_chiller_4 + Sequence.Q2kW_chiller_5 + Sequence.Q2kW_chiller_6;
Tot_Q2:=Chiller_1.Chiller_capacity_kW + Chiller_2.Chiller_capacity_kW + Chiller_3.Chiller_capacity_kW + Chiller_4.Chiller_capacity_kW (*+ Chiller_5.Chiller_capacity_kW + Chiller_6.Chiller_capacity_kW*);
COP_chiller_1:=Chiller_1.COP_chiller_ele;
COP_chiller_2:=Chiller_2.COP_chiller_ele;
COP_chiller_3:=Chiller_3.COP_chiller_ele;
COP_chiller_4:=Chiller_4.COP_chiller_ele;
(*COP_chiller_5:=Chiller_5.COP_chiller_ele;
COP_chiller_6:=Chiller_6.COP_chiller_ele;*)

totRunningChillers := BOOL_TO_INT(Chiller_1.Unit_running) + BOOL_TO_INT(Chiller_2.Unit_running) + BOOL_TO_INT(Chiller_3.Unit_running) + BOOL_TO_INT(Chiller_4.Unit_running)(* + BOOL_TO_INT(Chiller_5.Unit_running) + BOOL_TO_INT(Chiller_6.Unit_running)*);

IF Chiller_1.Unit_running THEN
	PI_calculation(Chiller_1.Chiller_capacity,Chiller_1.Temp_water_inlet_cond,COP_chiller_1,Chiller_1.Temp_chilled_medium_out, 1, PI_act=>PI_chiller_1, noCalc_error=>PI_Calc_Error_AC1, COP_theo=>COP_theo_AC1);	
	WastedEnergy_AC1 := Wasted_calc(Chiller_1.Chiller_capacity_kW, COP_theo_AC1, Power_motor_1_kW) ;
	ELSE
	PI_chiller_1 := 0;
	WastedEnergy_AC1 := 0;
	PI_Calc_Error_AC1 := TRUE;
	COP_theo_AC1 := 0;
END_IF

IF Chiller_2.Unit_running THEN
	PI_calculation(Chiller_2.Chiller_capacity,Chiller_2.Temp_water_inlet_cond,COP_chiller_2,Chiller_2.Temp_chilled_medium_out, 2, PI_act=>PI_chiller_2,noCalc_error=>PI_Calc_Error_AC2, COP_theo=>COP_theo_AC2);
	WastedEnergy_AC2 := Wasted_calc(Chiller_2.Chiller_capacity_kW, COP_theo_AC2, Power_motor_2_kW) ;
	ELSE
	PI_chiller_2 := 0;
	WastedEnergy_AC2 := 0;
	PI_Calc_Error_AC2 := TRUE;
	COP_theo_AC2 := 0;
END_IF

IF Chiller_3.Unit_running THEN
	PI_calculation(Chiller_3.Chiller_capacity,Chiller_3.Temp_water_inlet_cond,COP_chiller_3,Chiller_3.Temp_chilled_medium_out, 1, PI_act=>PI_chiller_3,noCalc_error=>PI_Calc_Error_AC3, COP_theo=>COP_theo_AC3);
	WastedEnergy_AC3 := Wasted_calc(Chiller_3.Chiller_capacity_kW, COP_theo_AC3, Power_motor_3_kW) ;
	ELSE
	PI_chiller_3 := 0;
	WastedEnergy_AC3 := 0;	
	PI_Calc_Error_AC3 := TRUE;
	COP_theo_AC3 := 0;
END_IF

IF Chiller_4.Unit_running THEN
	PI_calculation(Chiller_4.Chiller_capacity,Chiller_4.Temp_water_inlet_cond,COP_chiller_4,Chiller_4.Temp_chilled_medium_out, 2, PI_act=>PI_chiller_4,noCalc_error=>PI_Calc_Error_AC4, COP_theo=>COP_theo_AC4);
	WastedEnergy_AC4 := Wasted_calc(Chiller_4.Chiller_capacity_kW, COP_theo_AC4, Power_motor_4_kW) ;
	ELSE
	PI_chiller_4 := 0;
	WastedEnergy_AC4 := 0;
	PI_Calc_Error_AC4 := TRUE;
	COP_theo_AC4 := 0;
END_IF
(*
IF Chiller_5.Unit_running THEN
	PI_calculation(Chiller_5.Chiller_capacity,Chiller_5.Temp_water_inlet_cond,COP_chiller_5,Chiller_5.Temp_chilled_medium_out, 4, PI_act=>PI_chiller_5,noCalc_error=>PI_Calc_Error_AC5, COP_theo=>COP_theo_AC5);
	WastedEnergy_AC5 := Wasted_calc(sequence.Q2kW_chiller_5, COP_theo_AC5, Power_motor_5_kW) ;
	ELSE
	PI_chiller_5 := 0;
	WastedEnergy_AC5 := 0;
	PI_Calc_Error_AC5 := TRUE ;			
END_IF


IF Chiller_6.Unit_running THEN
	PI_calculation(Chiller_6.Chiller_capacity,Chiller_6.Temp_water_inlet_cond,COP_chiller_6,Chiller_6.Temp_chilled_medium_out, 2, PI_act=>PI_chiller_6,noCalc_error=>PI_Calc_Error_AC6, COP_theo=>COP_theo_AC6);
	WastedEnergy_AC6 := Wasted_calc(sequence.Q2kW_chiller_6, COP_theo_AC6, Power_motor_6_kW) ;
	ELSE
	PI_chiller_6 := 0;
	WastedEnergy_AC6 := 0 ;
	PI_Calc_Error_AC6 := TRUE ;			
END_IF
*)


PI_chiller_1_word := REAL_TO_WORD(PI_chiller_1 * 100) ;
PI_chiller_2_word := REAL_TO_WORD(PI_chiller_2 * 100) ;
PI_chiller_3_word := REAL_TO_WORD(PI_chiller_3 * 100) ;
PI_chiller_4_word := REAL_TO_WORD(PI_chiller_4 * 100) ;
//PI_chiller_5_word := REAL_TO_WORD(PI_chiller_5 * 100) ;
//PI_chiller_6_word := REAL_TO_WORD(PI_chiller_6 * 100) ;

WastedEnergy_AC1_word := REAL_TO_WORD(WastedEnergy_AC1) ;
WastedEnergy_AC2_word := REAL_TO_WORD(WastedEnergy_AC2) ;
WastedEnergy_AC3_word := REAL_TO_WORD(WastedEnergy_AC3) ;
WastedEnergy_AC4_word := REAL_TO_WORD(WastedEnergy_AC4) ;
//WastedEnergy_AC5_word := REAL_TO_WORD(WastedEnergy_AC5) ;
//WastedEnergy_AC6_word := REAL_TO_WORD(WastedEnergy_AC6) ;



(*
PI_calculation(95,31,4.5,6.1, 1, PI_act=>PI_chiller_1 ,noCalc_error=>PI_Calc_Error_AC1, COP_theo=>COP_theo_AC1);
PI_calculation(92,31,4.5,6.1, 3, PI_act=>PI_chiller_2 ,noCalc_error=>PI_Calc_Error_AC2, COP_theo=>COP_theo_AC2);
PI_calculation(91,31,4.5,6.1, 2, PI_act=>PI_chiller_3 ,noCalc_error=>PI_Calc_Error_AC3, COP_theo=>COP_theo_AC3);
PI_calculation(90,31,4.5,6.1, 3, PI_act=>PI_chiller_4 ,noCalc_error=>PI_Calc_Error_AC4, COP_theo=>COP_theo_AC4);
*)

IF totRunningChillers>0 THEN
	Total_PI:=Tot_PI(PI_chiller_1, PI_chiller_2, PI_chiller_3, PI_chiller_4, PI_chiller_5, PI_chiller_6 , totRunningChillers) ;
	ELSE 
	Total_PI := 0 ;
END_IF

END_PROGRAM

// csvRead
// CSV Reader examples
PROGRAM csvRead
VAR

	
	// 'ReadAll' example
	csvReaderInit3			: CSV.CSVReaderInit;
	csvReaderInit3COP		: CSV.CSVReaderInit;
	csvReaderInit3_1		: CSV.CSVReaderInit;
	csvReaderInit3_2		: CSV.CSVReaderInit;
	csvReaderInit3_3		: CSV.CSVReaderInit;
	xRead				: BOOL;
	xRead1				: BOOL;
	xRead2				: BOOL;
	xRead3				: BOOL;
	xReadCOP			: BOOL;
	readAll				: CSV.ReadAll;
	readAllCOP	    	: CSV.ReadAll;
	//COP Adj Array	
	// {attribute 'ac_persist' := 'PersistenceChannel'}
	// saDataArray			: ARRAY[0..8, 0..80] OF STRING(100);
	asDataArray			: ARRAY[0..730] OF STRING(100);
	pasDataArray		: POINTER TO ARRAY[0..730] OF STRING(100) := ADR(asDataArray);
	asDataArray1		: ARRAY[0..730] OF STRING(100);
	pasDataArray1		: POINTER TO ARRAY[0..730] OF STRING(100) := ADR(asDataArray1);
	asDataArray2		: ARRAY[0..730] OF STRING(100);
	pasDataArray2		: POINTER TO ARRAY[0..730] OF STRING(100) := ADR(asDataArray2);
	asDataArray3		: ARRAY[0..730] OF STRING(100);
	pasDataArray3		: POINTER TO ARRAY[0..730] OF STRING(100) := ADR(asDataArray3);
	//COP Adj Array
	// {attribute 'ac_persist' := 'PersistenceChannel'}
	// saCOPDataArray			: ARRAY[0..2, 0..320] OF STRING(100);
	asCOPDataArray		: ARRAY[0..970] OF STRING(100);
	pasCOPDataArray		: POINTER TO ARRAY[0..970] OF STRING(100) := ADR(asCOPDataArray);
	//  General variables
	dataConvert			: ConvertDataArray;
	dataConvert1		: ConvertDataArray_1;
	dataConvert2		: ConvertDataArray_2;
	dataConvert3		: ConvertDataArray_3;
	dataConvert4		: ConvertDataArray_4;
	R_TRIG_0			: R_TRIG;
	R_TRIG_1			: R_TRIG;
	R_TRIG_2			: R_TRIG;
	R_TRIG_3			: R_TRIG;
	R_TRIG_4			: R_TRIG;
	{attribute 'ac_persist' := 'PersistenceChannel'}
	PIfilename1			: STRING := '/home/jci/PIcsvfiles/NB6251_2400_VSD.csv' ;
	{attribute 'ac_persist' := 'PersistenceChannel'}
	PIfilename2			: STRING := '/home/jci/PIcsvfiles/NB6251_2400_DOL.csv' ;
	{attribute 'ac_persist' := 'PersistenceChannel'}
	PIfilename3			: STRING := '/home/jci/PIcsvfiles/' ;
	{attribute 'ac_persist' := 'PersistenceChannel'}
	PIfilename4			: STRING := '/home/jci/PIcsvfiles/' ;
	{attribute 'ac_persist' := 'PersistenceChannel'}
	copAdjfilename		: STRING := '/home/jci/PIcsvfiles/COP_adj.csv' ;
	initRead			: BOOL:= FALSE ;
	convFinished		: BOOL:= FALSE ;
	
END_VAR

// Read COP adj csv file
csvReaderInit3COP(xExecute := GVL.initRead, szFileName := copAdjfilename, sLineSeparator := '$L'); // CSV.CSVReaderInit
// Convert the data array for the visualization
// Convert the data array for the visualization
readAllCOP(
    xExecute := csvReaderInit3COP.xDone AND GVL.xReadCOP,
    udiMaxElementLength := 100,
    csvReaderInit := csvReaderInit3COP,
    pasDataArray := pasCOPDataArray); // CSV.ReadAll
R_TRIG_1(CLK := readAllCOP.xDone); // R_TRIG
dataConvert1(xExecute := R_TRIG_1.Q, asData := asCOPDataArray); // ConvertDataArray_1
// Read PI file
csvReaderInit3(xExecute := GVL.initRead, szFileName := PIfilename1, sLineSeparator := '$L'); // CSV.CSVReaderInit
readAll(
    xExecute := csvReaderInit3.xDone AND GVL.xRead,
    udiMaxElementLength := 100,
    csvReaderInit := csvReaderInit3,
    pasDataArray := pasDataArray); // CSV.ReadAll
GVL.saCOPDataArray := dataConvert1.asConvertedCOPData;
R_TRIG_0(CLK := readAll.xDone); // R_TRIG
dataConvert(xExecute := R_TRIG_0.Q, asData := asDataArray); // ConvertDataArray
// Read PI file4
csvReaderInit3_3(xExecute := GVL.initRead, szFileName := PIfilename4, sLineSeparator := '$L'); // CSV.CSVReaderInit
// Convert the data array for the visualization
// Convert the data array for the visualization
readAll(
    xExecute := csvReaderInit3_3.xDone AND GVL.xRead3,
    udiMaxElementLength := 100,
    csvReaderInit := csvReaderInit3_3,
    pasDataArray := pasDataArray3); // CSV.ReadAll
R_TRIG_4(CLK := readAll.xDone); // R_TRIG
dataConvert4(xExecute := R_TRIG_4.Q, asData := asDataArray3); // ConvertDataArray_4
GVL.saDataArray3 := dataConvert4.asConvertedData;
// Convert the data array for the visualization
convFinished := dataConvert1.convert_finished;
// Read PI file3
csvReaderInit3_2(xExecute := GVL.initRead, szFileName := PIfilename3, sLineSeparator := '$L'); // CSV.CSVReaderInit
// Convert the data array for the visualization
// Convert the data array for the visualization
readAll(
    xExecute := csvReaderInit3_2.xDone AND GVL.xRead2,
    udiMaxElementLength := 100,
    csvReaderInit := csvReaderInit3_2,
    pasDataArray := pasDataArray2); // CSV.ReadAll
R_TRIG_3(CLK := readAll.xDone); // R_TRIG
dataConvert3(xExecute := R_TRIG_3.Q, asData := asDataArray2); // ConvertDataArray_3
GVL.saDataArray2 := dataConvert3.asConvertedData;
// Read PI file 2
csvReaderInit3_1(xExecute := GVL.initRead, szFileName := PIfilename2, sLineSeparator := '$L'); // CSV.CSVReaderInit
// Convert the data array for the visualization
readAll(
    xExecute := csvReaderInit3_1.xDone AND GVL.xRead1,
    udiMaxElementLength := 100,
    csvReaderInit := csvReaderInit3_1,
    pasDataArray := pasDataArray1); // CSV.ReadAll
R_TRIG_2(CLK := readAll.xDone); // R_TRIG
dataConvert2(xExecute := R_TRIG_2.Q, asData := asDataArray1); // ConvertDataArray_2
GVL.saDataArray1 := dataConvert2.asConvertedData;
GVL.saDataArray := dataConvert.asConvertedData;

END_PROGRAM

// AC_DataLogManager
//Code generated by Application Composer.
//Modifying generated code is not recommended!
FUNCTION_BLOCK AC_DataLogManager EXTENDS AC_DataLog.DataLogManager
VAR_INPUT 
    INST_DataLogChannel : AC_DataLogManager_DataLogChannel;
    INST_DataLogChannel_1 : AC_DataLogManager_DataLogChannel_1;
    INST_DataLogChannel_2 : AC_DataLogManager_DataLogChannel_2;
    INST_DataLogChannel_3 : AC_DataLogManager_DataLogChannel_3;
    INST_DataLogChannel_4 : AC_DataLogManager_DataLogChannel_4;
    AC_ARRAY_pitfDataLogChannels : ARRAY[0..4] OF AC_DataLog.IDataLogChannel;
END_VAR

//Code generated by Application Composer.
//Modifying generated code is not recommended!
SUPER^();

END_FUNCTION_BLOCK

// /AC_Plant_Overview
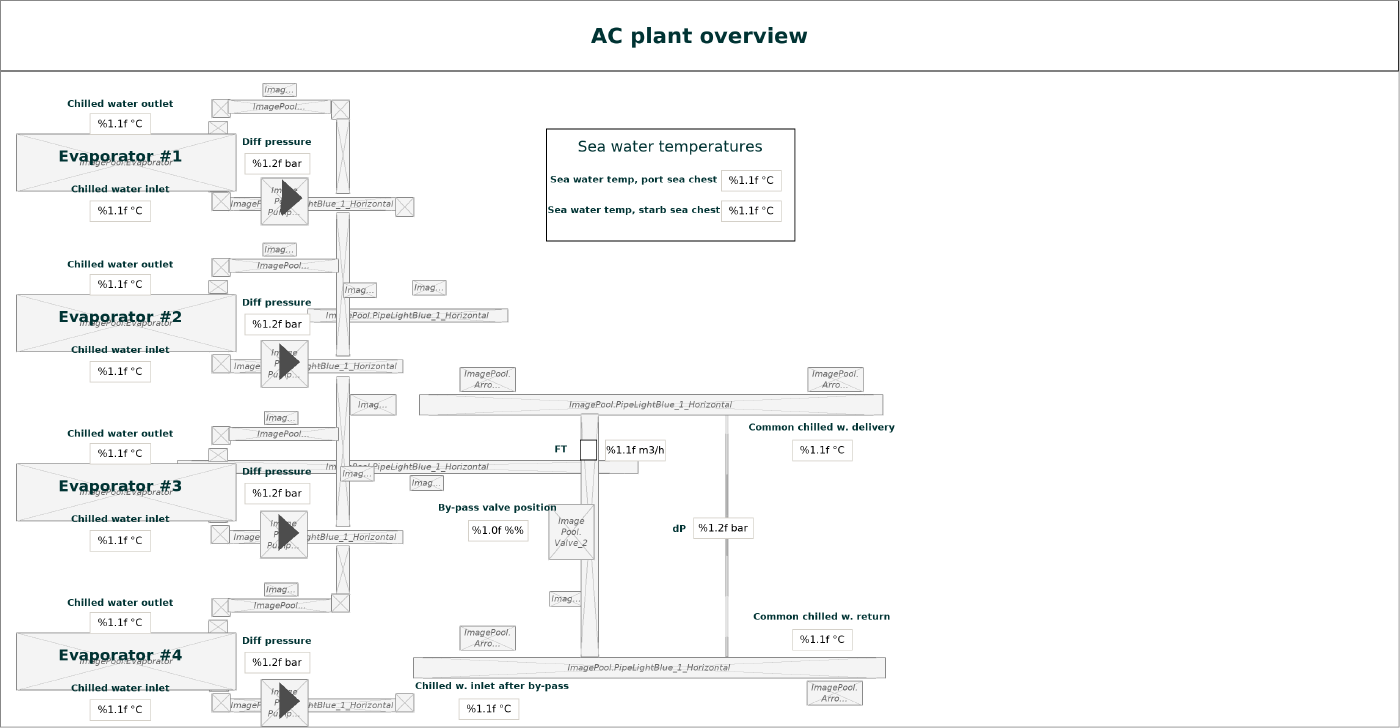
VISUALIZATION AC_Plant_Overview  // 1654x861
    Image (857,489 3x288), angle 180, image: ImagePool.PipeLightBlue_1_Vertical
    Image (209,544 545x16), angle 90, image: ImagePool.PipeLightBlue_1_Horizontal
    Image (363,365 237x16), angle 90, image: ImagePool.PipeLightBlue_1_Horizontal
    Image (246,143 23x16), angle 90, image: ImagePool.PipeLightBlue_1_Horizontal
    Rectangle (0,0 1652x84)
    Label (295,7 1063x70), "AC plant overview"
    Image (495,466 548x25), image: ImagePool.PipeLightBlue_1_Horizontal
    Image (270,233 198x16), image: ImagePool.PipeLightBlue_1_Horizontal
    Image (250,227 22x22), image: ImagePool.PipeLightBlue_3_RU
    Image (246,211 24x16), angle 270, image: ImagePool.PipeLightBlue_1_Horizontal
    Image (391,118 22x23), angle 90, image: ImagePool.PipeLightBlue_3_RD
    Image (19,158 260x68), image: ImagePool.Evaporator
    Label (65,165 155x40), "Evaporator #1"
    Label (285,153 84x30), "Diff pressure"
    Textfield (289,181 77x25), "%1.2f bar", text variable: Chiller_1.dP_CW
        p4168582468: Chiller_1.dP_CW
    Textfield (106,237 72x25), "%1.1f °C", text variable: Chiller_1.Temp_chilled_medium_in
        p4168582468: Chiller_1.Temp_chilled_medium_in
    Label (82,212 121x24), "Chilled water inlet"
    Image (308,210 56x56), image: ImagePool.Pump_Large_3
    Polygon (333,231) (333,212) (357,234) (333,255) (331,249), colour toggle: Chiller_1.DI_1_3
    Image (954,434 66x29), angle 180, image: ImagePool.Arrow lightblue left
    Image (953,805 66x29), image: ImagePool.Arrow lightblue left
    Image (649,699 40x18), angle 270, image: ImagePool.Arrow lightblue left
    Textfield (106,134 72x25), "%1.1f °C", text variable: Chiller_1.Temp_chilled_medium_out
        p4168582468: Chiller_1.Temp_chilled_medium_out
    Label (82,111 121x24), "Chilled water outlet"
    Image (246,331 23x16), angle 90, image: ImagePool.PipeLightBlue_1_Horizontal
    Image (270,425 206x16), image: ImagePool.PipeLightBlue_1_Horizontal
    Image (250,419 22x22), image: ImagePool.PipeLightBlue_3_RU
    Image (247,400 23x16), angle 270, image: ImagePool.PipeLightBlue_1_Horizontal
    Image (19,348 260x68), image: ImagePool.Evaporator
    Label (65,355 155x40), "Evaporator #2"
    Label (285,343 84x30), "Diff pressure"
    Textfield (289,371 77x25), "%1.2f bar", text variable: Chiller_2.dP_CW
        p4168582468: Chiller_2.dP_CW
    Textfield (106,427 72x25), "%1.1f °C", text variable: Chiller_2.Temp_chilled_medium_in
        p4168582468: Chiller_2.Temp_chilled_medium_in
    Label (82,402 121x24), "Chilled water inlet"
    Image (308,402 56x56), image: ImagePool.Pump_Large_3
    Polygon (330,425) (330,406) (354,428) (330,449) (330,441), colour toggle: Chiller_2.CW_Flow_ind
    Textfield (106,324 72x25), "%1.1f °C", text variable: Chiller_2.Temp_chilled_medium_out
        p4168582468: Chiller_2.Temp_chilled_medium_out
    Label (82,301 121x24), "Chilled water outlet"
    Image (246,530 23x16), angle 90, image: ImagePool.PipeLightBlue_1_Horizontal
    Image (269,627 207x16), image: ImagePool.PipeLightBlue_1_Horizontal
    Image (249,621 22x22), image: ImagePool.PipeLightBlue_3_RU
    Image (246,602 23x16), angle 270, image: ImagePool.PipeLightBlue_1_Horizontal
    Image (19,548 260x68), image: ImagePool.Evaporator
    Label (65,555 155x40), "Evaporator #3"
    Label (285,543 84x30), "Diff pressure"
    Textfield (289,571 77x25), "%1.2f bar", text variable: Chiller_3.dP_CW
        p4168582468: Chiller_3.dP_CW
    Textfield (106,627 72x25), "%1.1f °C", text variable: Chiller_3.Temp_chilled_medium_in
        p4168582468: Chiller_3.Temp_chilled_medium_in
    Label (82,602 121x24), "Chilled water inlet"
    Image (307,604 56x56), image: ImagePool.Pump_Large_3
    Polygon (329,627) (329,608) (353,630) (329,651) (329,643), colour toggle: Chiller_3.CW_Flow_ind
    Textfield (106,524 72x25), "%1.1f °C", text variable: Chiller_3.Temp_chilled_medium_out
        p4168582468: Chiller_3.Temp_chilled_medium_out
    Label (82,501 121x24), "Chilled water outlet"
    Image (246,733 23x16), angle 90, image: ImagePool.PipeLightBlue_1_Horizontal
    Image (270,826 198x16), image: ImagePool.PipeLightBlue_1_Horizontal
    Image (250,820 22x22), image: ImagePool.PipeLightBlue_3_RU
    Image (247,802 23x16), angle 270, image: ImagePool.PipeLightBlue_1_Horizontal
    Image (19,748 260x68), image: ImagePool.Evaporator
    Label (65,755 155x40), "Evaporator #4"
    Label (285,743 84x30), "Diff pressure"
    Textfield (289,771 77x25), "%1.2f bar", text variable: Chiller_4.dP_CW
        p4168582468: Chiller_4.dP_CW
    Textfield (106,827 72x25), "%1.1f °C", text variable: Chiller_4.Temp_chilled_medium_in
        p4168582468: Chiller_4.Temp_chilled_medium_in
    Label (82,802 121x24), "Chilled water inlet"
    Image (308,803 56x56), image: ImagePool.Pump_Large_3
    Polygon (330,826) (330,807) (354,829) (330,850) (330,842), colour toggle: Chiller_4.CW_Flow_ind
    Textfield (106,724 72x25), "%1.1f °C", text variable: Chiller_4.Temp_chilled_medium_out
        p4168582468: Chiller_4.Temp_chilled_medium_out
    Label (82,701 121x24), "Chilled water outlet"
    Textfield (936,520 71x25), "%1.1f °C", text variable: Sequence.Prim_CW_delivery_temp
        p4168582468: Sequence.Prim_CW_delivery_temp
    Image (397,645 16x58), angle 180, image: ImagePool.PipeLightBlue_1_Vertical
    Image (467,820 22x22), angle 90, image: ImagePool.PipeLightBlue_1_LD
    Image (467,233 22x23), angle 90, image: ImagePool.PipeLightBlue_3_RD
    Label (891,492 160x27), "Common chilled w. delivery"
    Image (250,117 22x22), angle 90, image: ImagePool.PipeLightBlue_3_RU
    Image (250,305 22x22), angle 90, image: ImagePool.PipeLightBlue_3_RU
    Image (250,504 22x22), angle 90, image: ImagePool.PipeLightBlue_3_RU
    Image (250,707 22x22), angle 90, image: ImagePool.PipeLightBlue_3_RU
    Image (269,708 124x16), image: ImagePool.PipeLightBlue_1_Horizontal
    Image (391,702 22x22), angle 90, image: ImagePool.PipeLightBlue_1_LD
    Image (397,445 16x178), angle 180, image: ImagePool.PipeLightBlue_1_Vertical
    Image (270,505 130x16), image: ImagePool.PipeLightBlue_1_Horizontal
    Image (269,118 122x16), image: ImagePool.PipeLightBlue_1_Horizontal
    Image (397,251 16x170), angle 180, image: ImagePool.PipeLightBlue_1_Vertical
    Image (270,306 130x16), image: ImagePool.PipeLightBlue_1_Horizontal
    Image (397,140 16x89), angle 180, image: ImagePool.PipeLightBlue_1_Vertical
    Image (488,777 558x25), image: ImagePool.PipeLightBlue_1_Horizontal
    Image (413,466 55x25), image: ImagePool.PipeLightBlue_1_Horizontal
    Image (686,489 21x288), angle 180, image: ImagePool.PipeLightBlue_1_Vertical
    Rectangle (645,152 294x133)
    Label (645,140 294x67), "Sea water temperatures"
    Image (648,596 54x66), angle 270, image: ImagePool.Valve_2
    Textfield (936,744 71x25), "%1.1f °C", text variable: Sequence.Prim_CW_return_temp
        p4168582468: Sequence.Prim_CW_return_temp
    Label (891,716 160x27), "Common chilled w. return"
    Textfield (542,826 71x25), "%1.1f °C", text variable: Sequence.Sec_CW_return_afterBP_temp
        p4168582468: Sequence.Sec_CW_return_afterBP_temp
    Label (497,798 169x27), "Chilled w. inlet after by-pass"
    Textfield (553,615 71x25), "%1.0f %%", text variable: Sequence.CW_Bypass_valve_FeedB
        p4168582468: Sequence.CW_Bypass_valve_FeedB
    Label (508,587 160x27), "By-pass valve position"
    Image (543,740 66x29), image: ImagePool.Arrow lightblue left
    Textfield (819,612 71x25), "%1.2f bar", text variable: Sequence.CW_dP_pumps
        p4168582468: Sequence.CW_dP_pumps
    Label (784,612 37x27), "dP"
    Image (543,434 66x29), angle 180, image: ImagePool.Arrow lightblue left
    Textfield (852,201 71x25), "%1.1f °C", text variable: Sequence.SW_temp_PS
        p4168582468: Sequence.SW_temp_PS
    Label (656,199 186x27), "Sea water temp, port sea chest"
    Textfield (852,237 71x25), "%1.1f °C", text variable: Sequence.SW_temp_SB
        p4168582468: Sequence.SW_temp_SB
    Label (656,235 186x27), "Sea water temp, starb sea chest"
    Image (487,331 40x18), angle 90, image: ImagePool.Arrow lightblue left
    Image (402,551 40x18), angle 90, image: ImagePool.Arrow lightblue left
    Image (484,562 40x18), angle 90, image: ImagePool.Arrow lightblue left
    Image (405,334 40x18), angle 270, image: ImagePool.Arrow lightblue left
    Image (310,98 40x16), angle 180, image: ImagePool.Arrow lightblue left
    Image (310,287 40x16), angle 180, image: ImagePool.Arrow lightblue left
    Image (312,486 40x16), angle 180, image: ImagePool.Arrow lightblue left
    Image (312,689 40x16), angle 180, image: ImagePool.Arrow lightblue left
    Label (644,518 37x27), "FT"
    Textfield (715,520 71x25), "%1.1f m3/h", tooltip "Sequence.CW_flowmeter_bypass", text variable: Sequence.CW_flowmeter_bypass
        p4168582468: Sequence.CW_flowmeter_bypass
    Rectangle (685,520 20x24)
END_VISUALIZATION

// /Alarm_list
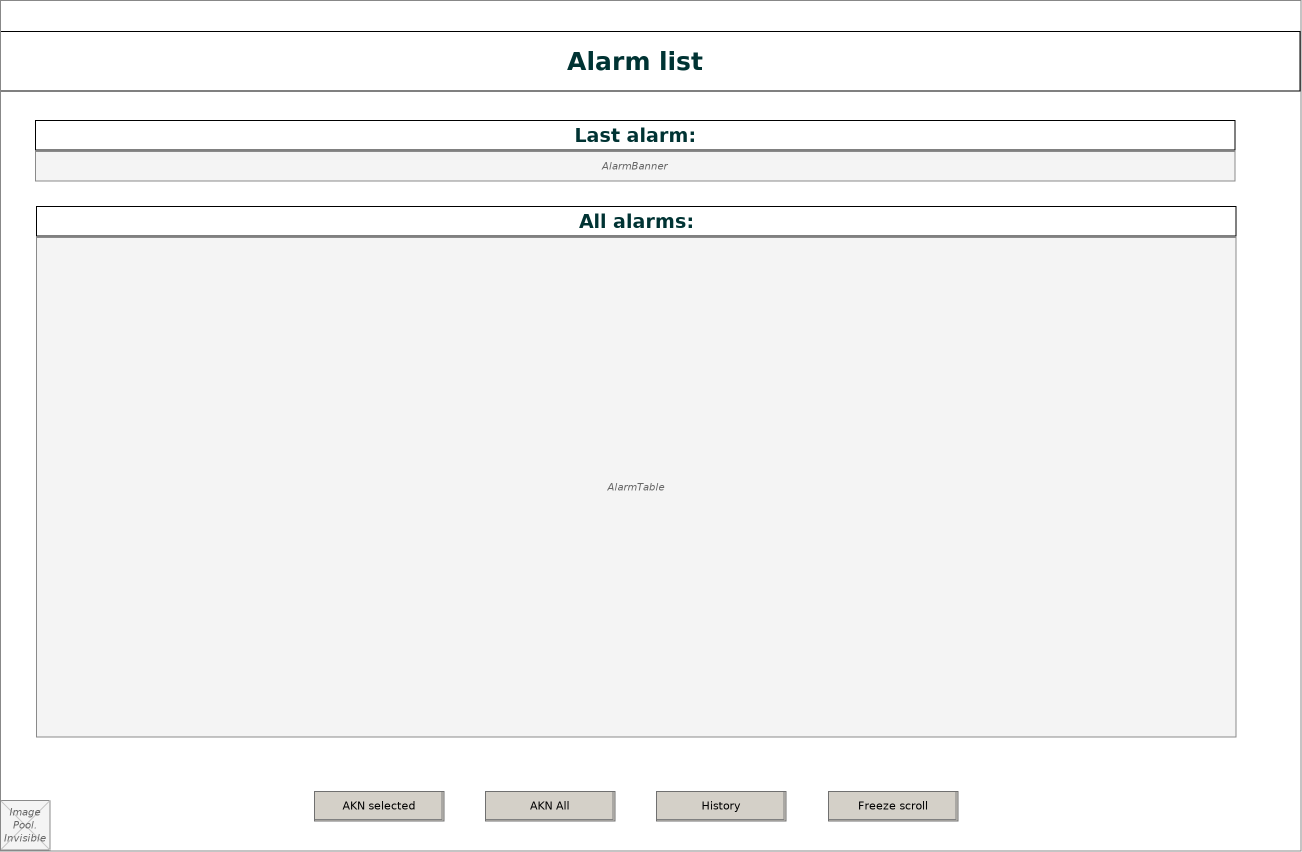
VISUALIZATION Alarm_list  // 1302x852
VAR
	AlarmACKButton : BOOL;
	AlarmACKAllButton : BOOL;
	AlarmHistoryButton : BOOL;
	AlarmFreezeButton : BOOL;
END_VAR
    AlarmTable (36,237 1200x500)
        p1521930926: __All
        p1663851261: __All
        p428520879: AlarmACKButton
        p2607059081: AlarmACKAllButton
        p3266827225: AlarmHistoryButton
        p3894972949: AlarmFreezeButton
    Button (314,791 130x30), "AKN selected"
        tap AlarmACKButton
    Button (485,791 130x30), "AKN All"
        tap AlarmACKAllButton
    Button (828,791 130x30), "Freeze scroll"
        toggle AlarmFreezeButton
    Button (656,791 130x30), "History"
        toggle AlarmHistoryButton
    Rectangle (0,31 1300x60)
    Label (247,33 776x56), "Alarm list"
    Rectangle (36,206 1200x30)
    Label (391,209 491x25), "All alarms:"
    Image (0,800 50x50), image: ImagePool.Invisible
    Rectangle (35,120 1200x30)
    Label (390,123 491x25), "Last alarm:"
    AlarmBanner (35,151 1200x30)
        p1521930926: __All
        p1663851261: __All
END_VISUALIZATION

// /Chiller1Menu
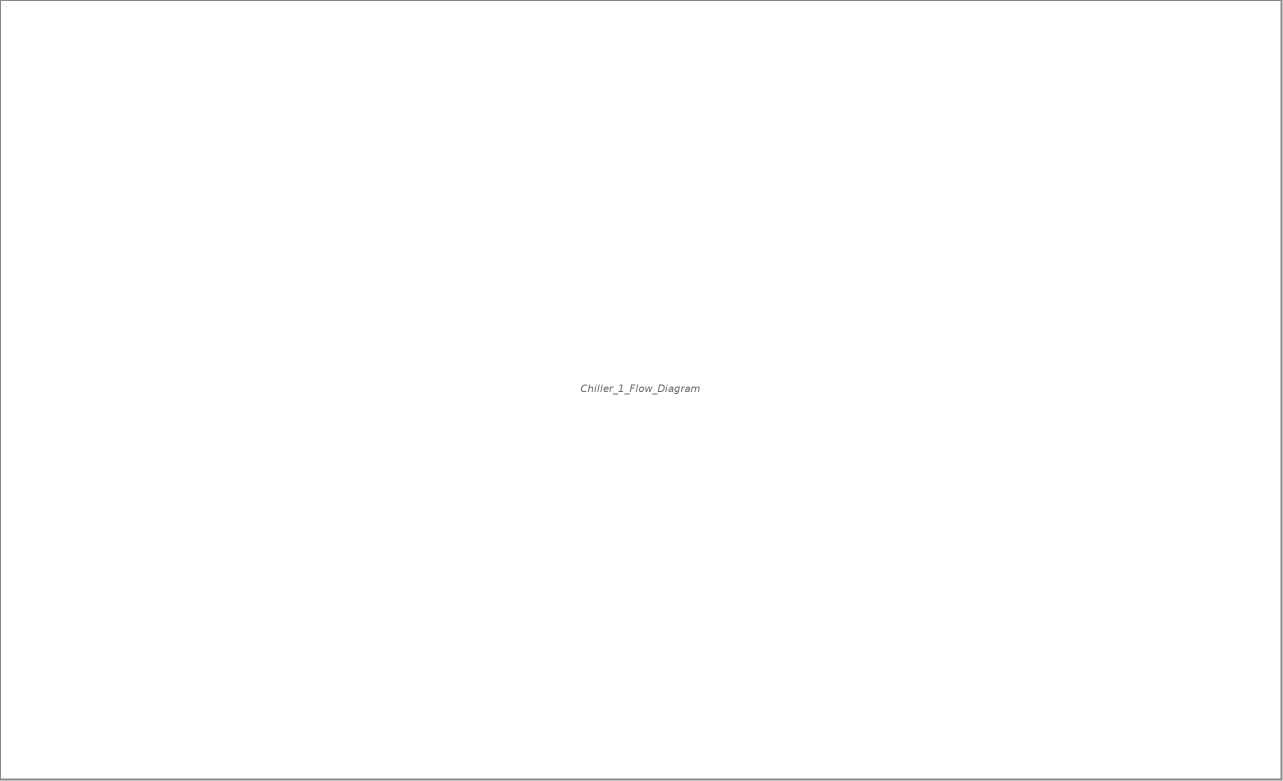
VISUALIZATION Chiller1Menu  // 1283x781
    TabControl (0,-2 1281x781)
        shows Chiller_1_Flow_Diagram()
        shows Chiller_1_Values()
        shows Chiller_1_Alarm()
        shows Chiller_1_Trip()
        shows Chiller_1_Oil()
        shows Chiller_1_VFD()
        shows TrendMenu()
        [0]: TabTitle=Diagram
        [1]: TabTitle=Measured values
        [2]: TabTitle=Alarm
        [3]: TabTitle=Trip
        [4]: TabTitle=Oil system
        [6]: TabTitle=Trend menu
END_VISUALIZATION

// /Chiller2Menu
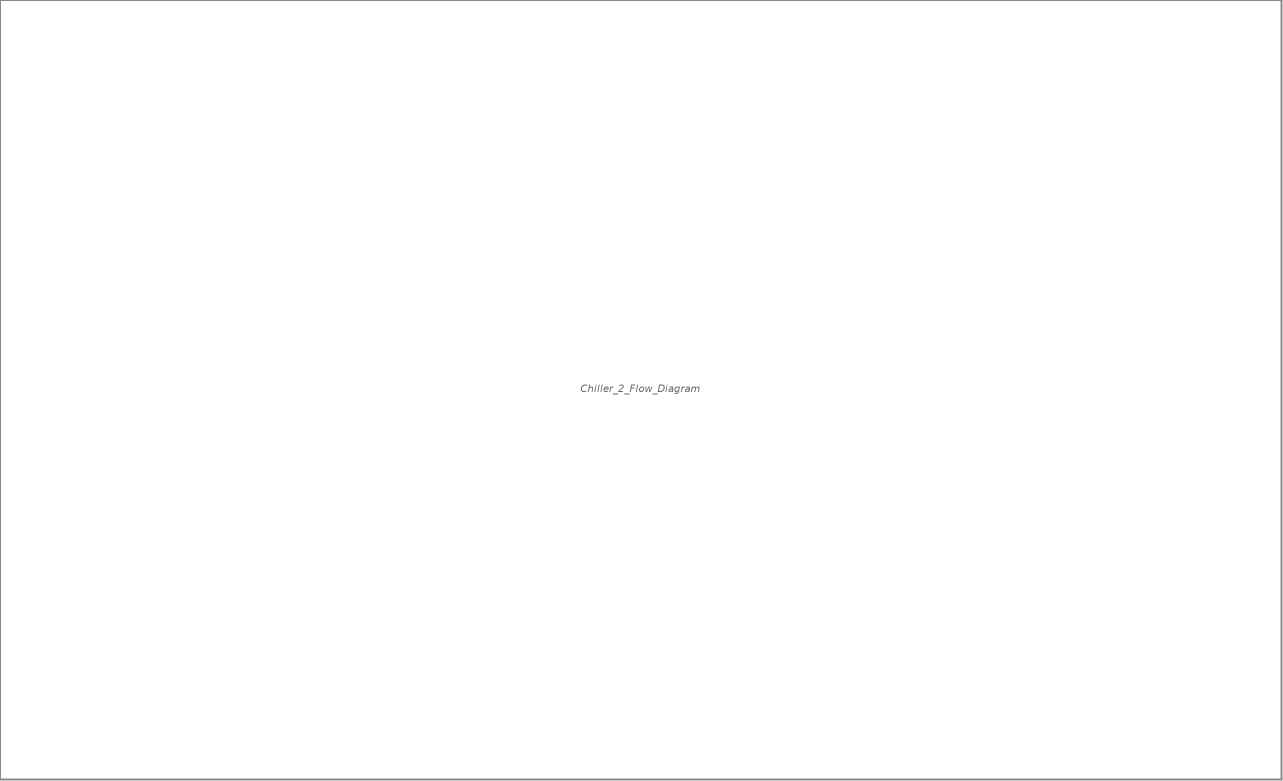
VISUALIZATION Chiller2Menu  // 1283x781
    TabControl (0,-2 1281x781)
        shows Chiller_2_Flow_Diagram()
        shows Chiller_2_Values()
        shows Chiller_2_Alarm()
        shows Chiller_2_Trip()
        shows Chiller_2_Oil()
        shows Chiller_1_Trip()
        [0]: TabTitle=Diagram
        [1]: TabTitle=Measured values
        [2]: TabTitle=Alarm
        [3]: TabTitle=Trip
        [4]: TabTitle=Oil system
        [5]: TabTitle=Trip
END_VISUALIZATION

// /Chiller3Menu
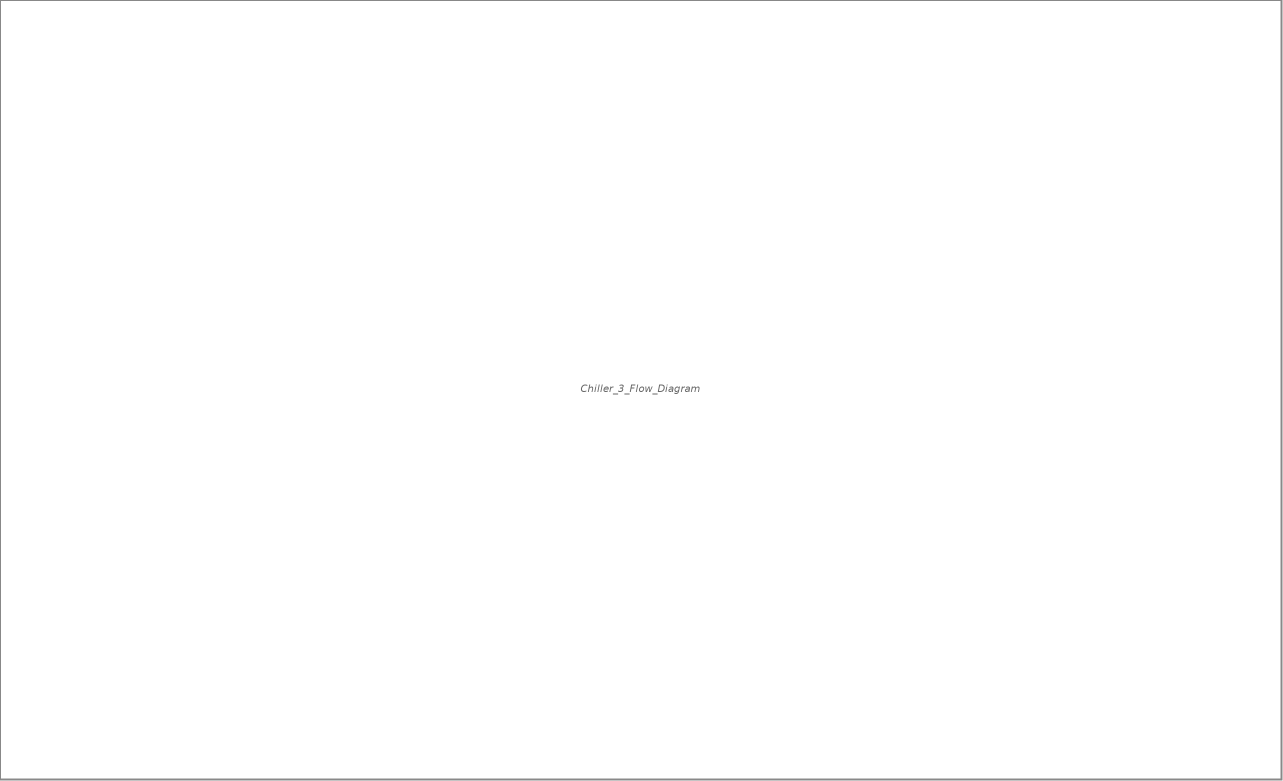
VISUALIZATION Chiller3Menu  // 1283x781
    TabControl (0,-2 1281x781)
        shows Chiller_3_Flow_Diagram()
        shows Chiller_3_Values()
        shows Chiller_3_Alarm()
        shows Chiller_3_Trip()
        shows Chiller_3_Oil()
        shows Chiller_3_VFD()
        [0]: TabTitle=Diagram
        [1]: TabTitle=Measured values
        [2]: TabTitle=Alarm
        [3]: TabTitle=Trip
        [4]: TabTitle=Oil system
END_VISUALIZATION

// /Chiller4Menu
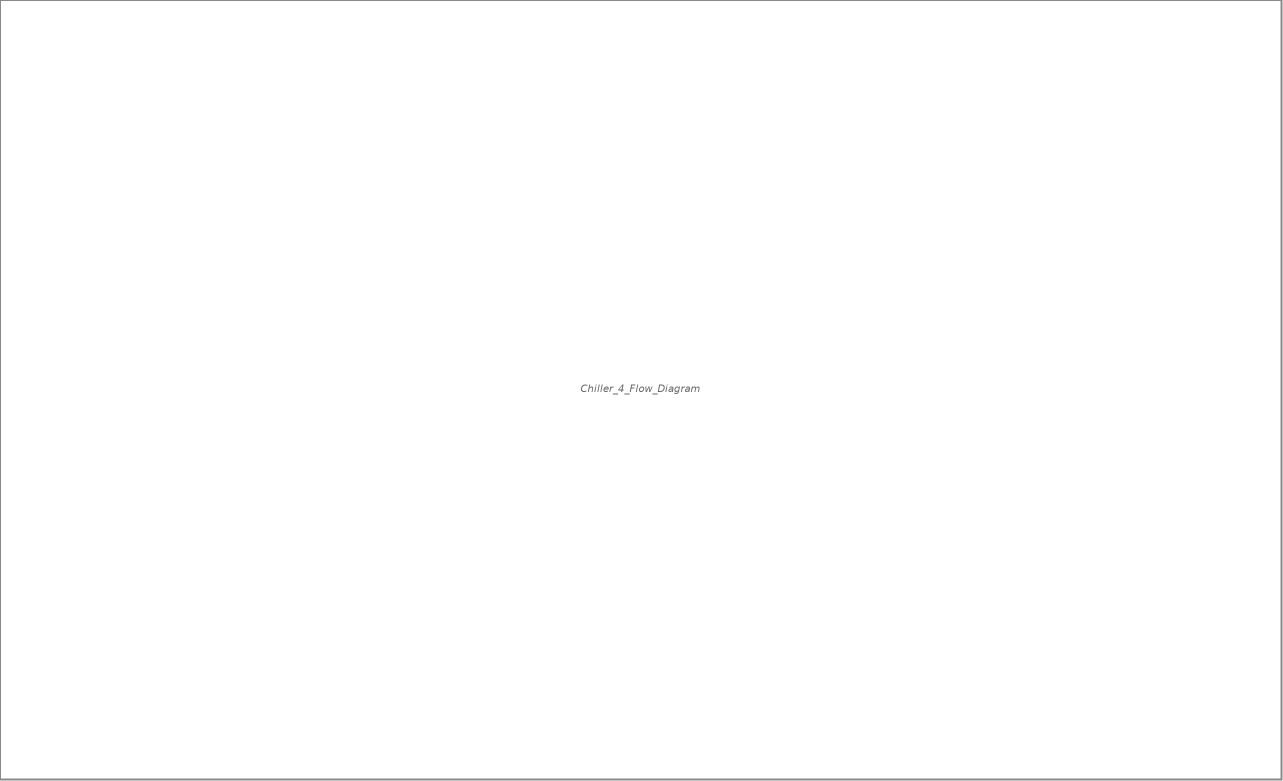
VISUALIZATION Chiller4Menu  // 1283x781
    TabControl (0,-2 1281x781)
        shows Chiller_4_Flow_Diagram()
        shows Chiller_4_Values()
        shows Chiller_4_Alarm()
        shows Chiller_4_Trip()
        shows Chiller_4_Oil()
        shows Chiller_1_Trip()
        [0]: TabTitle=Diagram
        [1]: TabTitle=Measured values
        [2]: TabTitle=Alarm
        [3]: TabTitle=Trip
        [4]: TabTitle=Oil system
        [5]: TabTitle=Trip
END_VISUALIZATION

// /Chiller_1_Alarm
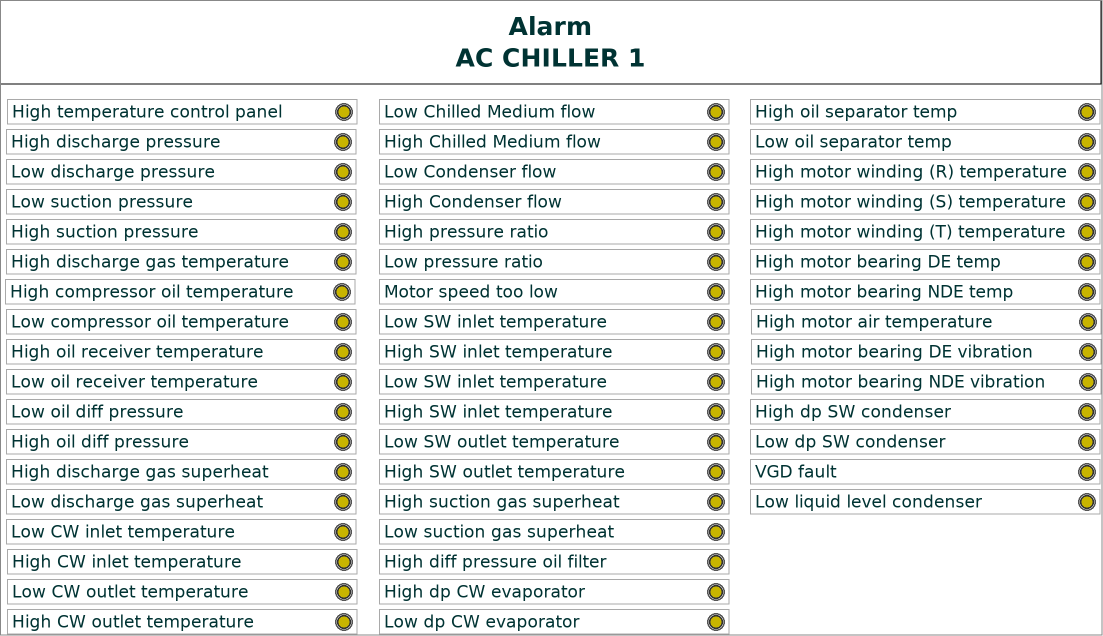
VISUALIZATION Chiller_1_Alarm  // 1103x636
    Rectangle (0,0 1101x84)
    Label (19,7 1063x70), "Alarm AC CHILLER 1"
    Rectangle (6,129 350x25)
    Label (8,131 318x21), "High discharge pressure"
    Lamp1 (332,132 22x20), variable: Chiller_1.A_high_disch_press, style: Lamp-Lamp1-Yellow
    Rectangle (6,189 350x25)
    Label (8,191 319x21), "Low suction pressure"
    Lamp1 (332,192 22x20), variable: Chiller_1.A_Low_suction_pressure, style: Lamp-Lamp1-Yellow
    Rectangle (6,219 350x25)
    Label (8,221 322x21), "High suction pressure"
    Lamp1 (332,222 22x20), variable: Chiller_1.A_High_suction_pressure, style: Lamp-Lamp1-Yellow
    Rectangle (6,249 350x25)
    Label (8,251 317x21), "High discharge gas temperature"
    Lamp1 (332,252 22x20), variable: Chiller_1.A_High_discharge_temp, style: Lamp-Lamp1-Yellow
    Rectangle (750,159 350x25)
    Label (752,161 320x21), "High motor winding (R) temperature"
    Lamp1 (1076,162 22x20), variable: Chiller_1.A_High_motor_wind_temp_R, style: Lamp-Lamp1-Yellow
    Rectangle (750,189 350x25)
    Label (752,191 319x21), "High motor winding (S) temperature"
    Lamp1 (1076,192 22x20), variable: Chiller_1.A_High_motor_wind_temp_S, style: Lamp-Lamp1-Yellow
    Rectangle (6,489 350x25)
    Label (8,491 319x21), "Low discharge gas superheat"
    Lamp1 (332,492 22x20), variable: Chiller_1.A_Low_discharge_superheat, style: Lamp-Lamp1-Yellow
    Rectangle (6,459 350x25)
    Label (8,461 322x21), "High discharge gas superheat"
    Lamp1 (332,462 22x20), variable: Chiller_1.A_High_discharge_superheat, style: Lamp-Lamp1-Yellow
    Rectangle (6,339 350x25)
    Label (8,341 317x21), "High oil receiver temperature"
    Lamp1 (332,342 22x20), variable: Chiller_1.A_High_oil_temp_receiver, style: Lamp-Lamp1-Yellow
    Rectangle (6,369 350x25)
    Label (8,371 319x21), "Low oil receiver temperature"
    Lamp1 (332,372 22x20), variable: Chiller_1.A_Low_oil_temp_receiver, style: Lamp-Lamp1-Yellow
    Rectangle (6,399 350x25)
    Label (8,401 322x21), "Low oil diff pressure"
    Lamp1 (332,402 22x20), variable: Chiller_1.A_Low_oil_diff_pressure, style: Lamp-Lamp1-Yellow
    Rectangle (6,429 350x25)
    Label (8,431 317x21), "High oil diff pressure"
    Lamp1 (332,432 22x20), variable: Chiller_1.A_High_oil_diff_pressure, style: Lamp-Lamp1-Yellow
    Rectangle (6,309 350x25)
    Label (8,311 319x21), "Low compressor oil temperature"
    Lamp1 (332,312 22x20), variable: Chiller_1.A_Low_temp_oil_inlet_comp, style: Lamp-Lamp1-Yellow
    Rectangle (5,279 350x25)
    Label (7,281 322x21), "High compressor oil temperature"
    Lamp1 (331,282 22x20), variable: Chiller_1.A_High_temp_oil_inlet_comp, style: Lamp-Lamp1-Yellow
    Rectangle (379,309 350x25)
    Label (381,311 317x21), "Low SW inlet temperature"
    Lamp1 (705,312 22x20), variable: Chiller_1.A_Low_SW_inlet_temp, style: Lamp-Lamp1-Yellow
    Rectangle (7,549 350x25)
    Label (9,551 322x21), "High CW inlet temperature"
    Lamp1 (333,552 22x20), variable: Chiller_1.A_High_CW_inlet_temp, style: Lamp-Lamp1-Yellow
    Rectangle (6,519 350x25)
    Label (8,521 317x21), "Low CW inlet temperature"
    Lamp1 (332,522 22x20), variable: Chiller_1.A_Low_CW_inlet_temp, style: Lamp-Lamp1-Yellow
    Rectangle (379,549 350x25)
    Label (381,551 317x21), "High diff pressure oil filter"
    Lamp1 (705,552 22x20), variable: Chiller_1.A_High_oil_filter_diff_press, style: Lamp-Lamp1-Yellow
    Rectangle (750,219 350x25)
    Label (752,221 317x21), "High motor winding (T) temperature"
    Lamp1 (1076,222 22x20), variable: Chiller_1.A_High_motor_wind_temp_T, style: Lamp-Lamp1-Yellow
    Rectangle (750,249 350x25)
    Label (752,251 317x21), "High motor bearing DE temp"
    Lamp1 (1076,252 22x20), variable: Chiller_1.A_High_comp_mo_DE_bear_temp, style: Lamp-Lamp1-Yellow
    Rectangle (750,279 350x25)
    Label (752,281 319x21), "High motor bearing NDE temp"
    Lamp1 (1076,282 22x20), variable: Chiller_1.A_High_comp_mo_NDE_bear_temp, style: Lamp-Lamp1-Yellow
    Rectangle (751,309 350x25)
    Label (753,311 322x21), "High motor air temperature"
    Lamp1 (1077,312 22x20), variable: Chiller_1.A_High_motor_air_temp, style: Lamp-Lamp1-Yellow
    Rectangle (751,339 350x25)
    Label (753,341 317x21), "High motor bearing DE vibration"
    Lamp1 (1077,342 22x20), variable: Chiller_1.A_High_comp_mo_DE_bear_vib, style: Lamp-Lamp1-Yellow
    Rectangle (751,369 350x25)
    Label (753,371 319x21), "High motor bearing NDE vibration"
    Lamp1 (1077,372 22x20), variable: Chiller_1.A_High_comp_mo_NDE_bear_vib, style: Lamp-Lamp1-Yellow
    Rectangle (379,579 350x25)
    Label (381,581 322x21), "High dp CW evaporator"
    Lamp1 (705,582 22x20), variable: Chiller_1.A_High_CW_dP, style: Lamp-Lamp1-Yellow
    Rectangle (379,609 350x25)
    Label (381,611 317x21), "Low dp CW evaporator"
    Lamp1 (705,612 22x20), variable: Chiller_1.A_Low_CW_dP, style: Lamp-Lamp1-Yellow
    Rectangle (750,399 350x25)
    Label (752,401 319x21), "High dp SW condenser"
    Lamp1 (1076,402 22x20), variable: Chiller_1.A_High_SW_dP, style: Lamp-Lamp1-Yellow
    Rectangle (750,429 350x25)
    Label (752,431 322x21), "Low dp SW condenser"
    Lamp1 (1076,432 22x20), variable: Chiller_1.A_Low_SW_dP, style: Lamp-Lamp1-Yellow
    Rectangle (750,459 350x25)
    Label (752,461 317x21), "VGD fault"
    Lamp1 (1076,462 22x20), variable: Chiller_1.A_VGD_Fault, style: Lamp-Lamp1-Yellow
    Rectangle (750,489 350x25)
    Label (752,491 317x21), "Low liquid level condenser"
    Lamp1 (1076,492 22x20), variable: Chiller_1.A_Low_liquid_level, style: Lamp-Lamp1-Yellow
    Rectangle (6,159 350x25)
    Label (8,161 318x21), "Low discharge pressure"
    Lamp1 (332,162 22x20), variable: Chiller_1.A_low_disch_press, style: Lamp-Lamp1-Yellow
    Rectangle (379,339 350x25)
    Label (381,341 314x21), "High SW inlet temperature"
    Lamp1 (705,342 22x20), variable: Chiller_1.A_High_SW_inlet_temp, style: Lamp-Lamp1-Yellow
    Rectangle (7,99 350x25)
    Label (9,101 318x21), "High temperature control panel"
    Lamp1 (333,102 22x20), variable: Chiller_1.A_low_disch_press, style: Lamp-Lamp1-Yellow
    Rectangle (7,579 350x25)
    Label (9,581 317x21), "Low CW outlet temperature"
    Lamp1 (333,582 22x20), variable: Chiller_1.A_Low_CW_outlet_temp, style: Lamp-Lamp1-Yellow
    Rectangle (7,609 350x25)
    Label (9,611 317x21), "High CW outlet temperature"
    Lamp1 (333,612 22x20), variable: Chiller_1.A_high_CW_outlet_temp, style: Lamp-Lamp1-Yellow
    Rectangle (379,99 350x25)
    Label (381,101 317x21), "Low Chilled Medium flow"
    Lamp1 (705,102 22x20), variable: Chiller_1.A_Low_chilled_medium_flow, style: Lamp-Lamp1-Yellow
    Rectangle (379,129 350x25)
    Label (381,131 317x21), "High Chilled Medium flow"
    Lamp1 (705,132 22x20), variable: Chiller_1.A_High_chilled_medium_flow, style: Lamp-Lamp1-Yellow
    Rectangle (379,159 350x25)
    Label (381,161 317x21), "Low Condenser flow"
    Lamp1 (705,162 22x20), variable: Chiller_1.A_Low_condenser_flow, style: Lamp-Lamp1-Yellow
    Rectangle (379,189 350x25)
    Label (381,191 317x21), "High Condenser flow"
    Lamp1 (705,192 22x20), variable: Chiller_1.A_High_condenser_flow, style: Lamp-Lamp1-Yellow
    Rectangle (379,219 350x25)
    Label (381,221 317x21), "High pressure ratio"
    Lamp1 (705,222 22x20), variable: Chiller_1.A_High_press_ratio, style: Lamp-Lamp1-Yellow
    Rectangle (379,249 350x25)
    Label (381,251 317x21), "Low pressure ratio"
    Lamp1 (705,252 22x20), variable: Chiller_1.A_Low_press_ratio, style: Lamp-Lamp1-Yellow
    Rectangle (379,279 350x25)
    Label (381,281 317x21), "Motor speed too low"
    Lamp1 (705,282 22x20), variable: Chiller_1.A_Motor_speed_low, style: Lamp-Lamp1-Yellow
    Rectangle (379,369 350x25)
    Label (381,371 317x21), "Low SW inlet temperature"
    Lamp1 (705,372 22x20), variable: Chiller_1.A_Low_SW_inlet_temp, style: Lamp-Lamp1-Yellow
    Rectangle (379,399 350x25)
    Label (381,401 314x21), "High SW inlet temperature"
    Lamp1 (705,402 22x20), variable: Chiller_1.A_High_SW_inlet_temp, style: Lamp-Lamp1-Yellow
    Rectangle (379,429 350x25)
    Label (381,431 317x21), "Low SW outlet temperature"
    Lamp1 (705,432 22x20), variable: Chiller_1.A_Low_SW_outlet_temp, style: Lamp-Lamp1-Yellow
    Rectangle (379,459 350x25)
    Label (381,461 314x21), "High SW outlet temperature"
    Lamp1 (705,462 22x20), variable: Chiller_1.A_High_SW_outlet_temp, style: Lamp-Lamp1-Yellow
    Rectangle (379,489 350x25)
    Label (381,491 317x21), "High suction gas superheat"
    Lamp1 (705,492 22x20), variable: Chiller_1.A_High_suction_superheat, style: Lamp-Lamp1-Yellow
    Rectangle (379,519 350x25)
    Label (381,521 314x21), "Low suction gas superheat"
    Lamp1 (705,522 22x20), variable: Chiller_1.A_Low_suction_superheat, style: Lamp-Lamp1-Yellow
    Rectangle (750,99 350x25)
    Label (752,101 317x21), "High oil separator temp"
    Lamp1 (1076,102 22x20), variable: Chiller_1.A_High_temp_oil_separator, style: Lamp-Lamp1-Yellow
    Rectangle (750,129 350x25)
    Label (752,131 319x21), "Low oil separator temp"
    Lamp1 (1076,132 22x20), variable: Chiller_1.A_Low_temp_oil_separator, style: Lamp-Lamp1-Yellow
END_VISUALIZATION

// /Chiller_1_Flow_Diagram
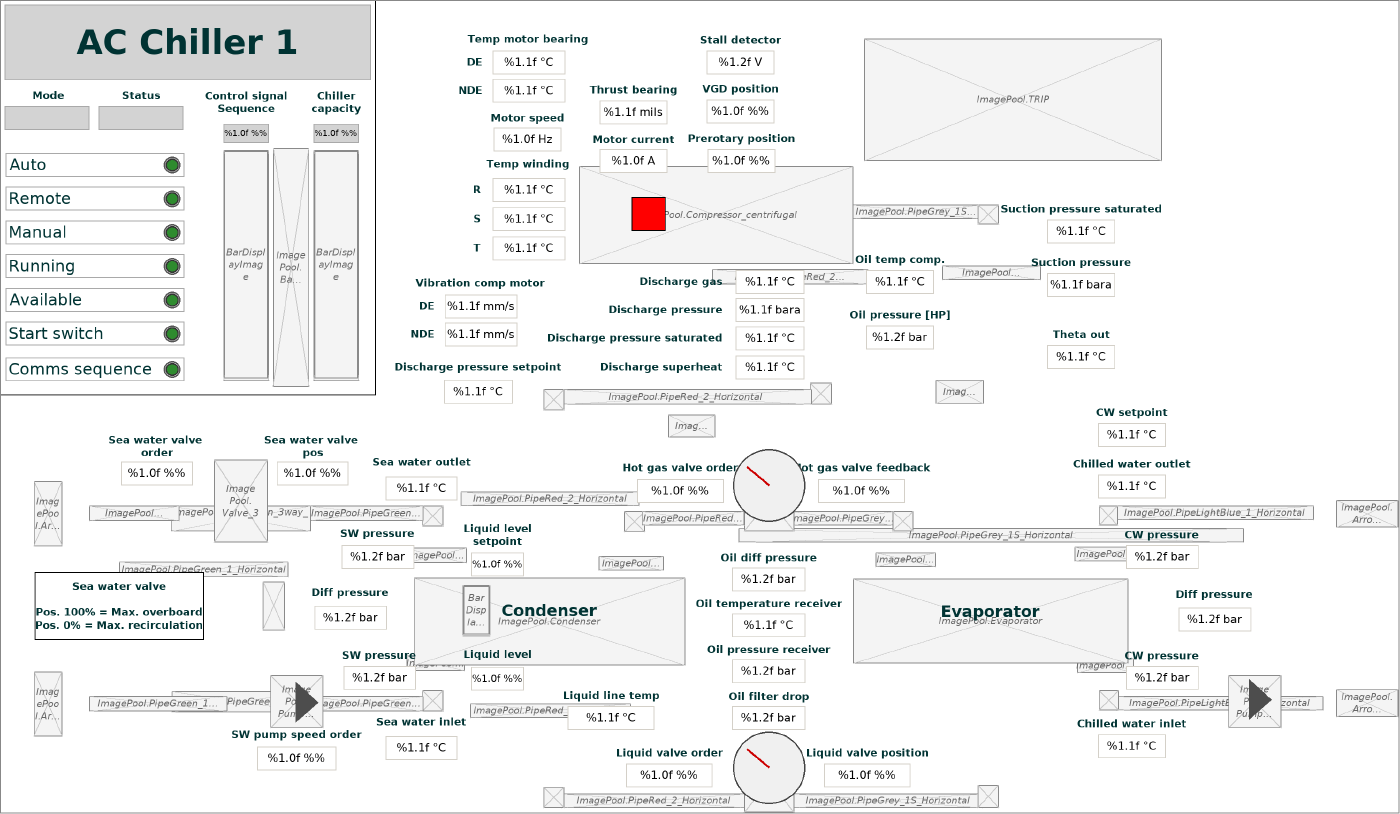
VISUALIZATION Chiller_1_Flow_Diagram  // 1492x868
    Rectangle (0,0 400x421)
    Textfield (238,132 48x20), "%1.0f %%", text variable: Sequence.Seq_cap_order_C1
        p4168582468: Sequence.Seq_cap_order_C1
    Image (1148,702 60x15), angle 270, image: ImagePool.PipeLightBlue_1_Horizontal
    Image (1145,583 67x15), angle 270, image: ImagePool.PipeLightBlue_1_Horizontal
    Image (908,218 137x15), image: ImagePool.PipeGrey_1S_Horizontal
    Image (845,846 202x15), image: ImagePool.PipeGrey_1S_Horizontal
    Image (933,589 64x15), angle 270, image: ImagePool.PipeGrey_1S_Horizontal
    Image (787,563 538x15), angle 270, image: ImagePool.PipeGrey_1S_Horizontal
    Image (843,545 110x15), image: ImagePool.PipeGrey_1S_Horizontal
    Image (638,593 69x15), angle 270, image: ImagePool.PipeRed_2_Horizontal
    Image (501,750 171x15), angle 270, image: ImagePool.PipeRed_2_Horizontal
    Label (218,94 89x30), "Control signal Sequence"
    Image (617,177 292x104), image: ImagePool.Compressor_centrifugal
    Image (759,287 166x16), angle 270, image: ImagePool.PipeRed_2_Horizontal
    Image (863,408 23x23), image: ImagePool.PipeRed_2_LU
    Image (596,415 269x16), image: ImagePool.PipeRed_2_Horizontal
    Image (909,617 293x90), image: ImagePool.Evaporator
    Image (431,584 66x16), angle 270, image: ImagePool.PipeGreen_1_Horizontal
    Image (450,539 22x22), image: ImagePool.PipeGreen_1_LD
    Image (329,539 122x16), image: ImagePool.PipeGreen_1_Horizontal
    Label (331,617 84x30), "Diff pressure"
    Textfield (335,646 77x25), "%1.2f bar", text variable: Chiller_1.dP_SW
        p4168582468: Chiller_1.dP_SW
    Image (127,599 180x16), angle 270, image: ImagePool.PipeGreen_1_Horizontal
    Image (183,737 147x22), image: ImagePool.PipeGreen_3way
    Image (433,699 62x16), angle 270, image: ImagePool.PipeGreen_1_Horizontal
    Image (450,736 22x22), image: ImagePool.PipeGreen_2_LU
    Image (329,742 122x16), image: ImagePool.PipeGreen_1_Horizontal
    Image (182,539 149x27), image: ImagePool.PipeGreen_3way_2
    Image (288,720 56x56), image: ImagePool.Pump_Large_3
    Polygon (315,746) (315,727) (339,749) (315,770) (315,762), colour toggle: Chiller_1.Sea_water_pump
    Image (36,513 30x69), angle 90, image: ImagePool.Arrow green down
    Image (36,716 30x69), angle 270, image: ImagePool.Arrow green down
    Image (579,415 22x22), image: ImagePool.PipeRed_1_RD
    Image (491,524 190x15), angle 270, image: ImagePool.PipeRed_2_Horizontal
    Label (360,554 84x30), "SW pressure"
    Textfield (364,581 77x25), "%1.2f bar", text variable: Chiller_1.Press_water_cond_out
        p4168582468: Chiller_1.Press_water_cond_out
    Image (95,539 96x16), image: ImagePool.PipeGreen_1_Horizontal
    Image (441,616 289x93), image: ImagePool.Condenser
    Image (598,846 197x15), image: ImagePool.PipeRed_2_Horizontal
    Image (579,839 22x22), image: ImagePool.PipeRed_2_RU
    Label (362,684 84x30), "SW pressure"
    Textfield (366,710 77x25), "%1.2f bar", text variable: Chiller_1.Press_water_cond_inlet
        p4168582468: Chiller_1.Press_water_cond_inlet
    Image (793,501 53x65), image: ImagePool.Valve_2
    Image (793,801 53x65), image: ImagePool.Valve_2
    Image (665,545 22x22), image: ImagePool.PipeRed_1_RD
    Image (684,545 109x15), image: ImagePool.PipeRed_2_Horizontal
    Image (951,545 22x21), image: ImagePool.PipeGrey_2_LD
    Image (1042,837 22x24), image: ImagePool.PipeGrey_3_LU
    Image (1042,218 22x21), image: ImagePool.PipeGrey_2_LD
    Image (1004,283 105x15), angle 270, image: ImagePool.PipeGrey_1S_Horizontal
    Label (521,636 129x30), "Condenser"
    Label (991,637 129x30), "Evaporator"
    Image (1189,539 211x15), image: ImagePool.PipeLightBlue_1_Horizontal
    Image (1171,539 20x21), image: ImagePool.PipeLightBlue_3_RD
    Image (1190,742 220x15), image: ImagePool.PipeLightBlue_1_Horizontal
    Image (1171,736 21x21), image: ImagePool.PipeLightBlue_3_RU
    Image (1424,533 66x29), angle 180, image: ImagePool.Arrow lightblue left
    Image (1424,735 66x29), image: ImagePool.Arrow lightblue left
    Image (1309,720 56x56), image: ImagePool.Pump_Large_3
    Polygon (1331,743) (1331,724) (1355,746) (1331,767) (1331,759), colour toggle: Chiller_1.CW_Flow_ind
    Image (280,620 23x52), image: ImagePool.Arrow green down
    Image (712,442 50x24), image: ImagePool.Arrow red left
    Image (997,405 51x25), angle 90, image: ImagePool.Arrow gray left
    Image (291,158 38x254), image: ImagePool.BarScale3
    Label (324,94 69x30), "Chiller capacity"
    Textfield (105,113 90x25), text list: 'TextList_PT', text index: Chiller_1.Unit_switch_status
    Textfield (5,113 90x25), text list: 'TextList_PT', text index: Chiller_1.Unit_start_switch
    Textfield (334,132 48x20), "%1.0f %%", text variable: Chiller_1.Chiller_capacity_t1
        p4168582468: Chiller_1.Chiller_capacity_t1
    Textfield (5,5 390x80), "AC Chiller 1"
    Label (521,160 84x30), "Temp winding"
    Textfield (525,190 77x25), "%1.1f °C", text variable: Chiller_1.Temp_motor_wind_R
        p4168582468: Chiller_1.Temp_motor_wind_R
    Label (496,190 25x25), "R"
    Textfield (525,221 77x25), "%1.1f °C", text variable: Chiller_1.Temp_motor_wind_S
        p4168582468: Chiller_1.Temp_motor_wind_S
    Label (496,221 25x25), "S"
    Textfield (525,252 77x25), "%1.1f °C", text variable: Chiller_1.Temp_motor_wind_T
        p4168582468: Chiller_1.Temp_motor_wind_T
    Label (496,252 25x25), "T"
    Textfield (679,511 92x25), "%1.0f %%", text variable: Chiller_1.Hot_gas_valve_output
        p4168582468: Chiller_1.Hot_gas_valve_output
    Label (664,484 122x30), "Hot gas valve order"
    Label (849,484 139x30), "Hot gas valve feedback"
    Textfield (872,511 92x25), "%1.0f %%", text variable: Chiller_1.Feedback_HGV
        p4168582468: Chiller_1.Feedback_HGV
    Meter360 (781,479 77x77), value: Chiller_1.Feedback_HGV, style: Meter-Meter360-Gray, scale format: %1.0f, scale 0..100
        p3451962224: ImagePool.Invisible
    Meter360 (781,780 77x77), value: Chiller_1.Feedback_liquid_valve, style: Meter-Meter360-Gray, scale format: %1.0f, scale 0..100
        p3451962224: ImagePool.Invisible
    Textfield (502,589 56x25), "%1.0f %%", text variable: Chiller_1.SP_PID_Level
        p4168582468: Chiller_1.SP_PID_Level
    Label (494,551 73x39), "Liquid level setpoint"
    Textfield (502,711 56x25), "%1.0f %%", text variable: Chiller_1.Liquid_level_condenser
        p4168582468: Chiller_1.Liquid_level_condenser
    Label (491,683 79x30), "Liquid level"
    Textfield (639,159 72x25), "%1.0f A", text variable: Chiller_1.Motor_current
        p4168582468: Chiller_1.Motor_current
    Label (634,138 83x22), "Motor current"
    Textfield (274,796 84x25), "%1.0f %%", text variable: Chiller_1.SW_pump_speed_order
        p4168582468: Chiller_1.SW_pump_speed_order
    Label (250,770 132x27), "SW pump speed order"
    Textfield (473,405 73x25), "%1.1f °C", tooltip "Chiller_1.SP_PID_seawater", text variable: Chiller_1.SP_PID_seawater
    Textfield (784,348 73x25), "%1.1f °C", text variable: Chiller_1.Discharge_saturated_temp
        p4168582468: Chiller_1.Discharge_saturated_temp
    Label (589,347 184x27), "Discharge pressure saturated"
    Label (425,378 169x27), "Discharge pressure setpoint"
    Textfield (411,785 76x25), "%1.1f °C", text variable: Chiller_1.Temp_water_inlet_cond
        p4168582468: Chiller_1.Temp_water_inlet_cond
    Label (399,755 100x30), "Sea water inlet"
    Textfield (411,508 76x25), "%1.1f °C", text variable: Chiller_1.Temp_water_outlet_cond
        p4168582468: Chiller_1.Temp_water_outlet_cond
    Label (397,478 105x30), "Sea water outlet"
    Label (500,27 126x30), "Temp motor bearing"
    Textfield (525,84 77x25), "%1.1f °C", text variable: Chiller_1.Temp_motor_bearing_NDE
        p4168582468: Chiller_1.Temp_motor_bearing_NDE
    Textfield (525,54 77x25), "%1.1f °C", text variable: Chiller_1.Temp_motor_bearing_DE
        p4168582468: Chiller_1.Temp_motor_bearing_DE
    Label (480,54 37x25), "DE"
    Label (480,84 37x25), "NDE"
    Label (678,287 95x27), "Discharge gas"
    Textfield (784,288 73x25), "%1.1f °C", text variable: Chiller_1.Temp_discharge
        p4168582468: Chiller_1.Temp_discharge
    Label (644,317 129x27), "Discharge pressure"
    Textfield (784,318 73x25), "%1.1f bara", text variable: Chiller_1.Press_discharge_compr
        p4168582468: Chiller_1.Press_discharge_compr
    Textfield (784,379 73x25), "%1.1f °C", text variable: Chiller_1.Discharge_superheat
        p4168582468: Chiller_1.Discharge_superheat
    Label (589,378 184x27), "Discharge superheat"
    Label (631,84 89x24), "Thrust bearing"
    Textfield (639,107 72x25), "%1.1f mils", text variable: Chiller_1.Thrust_bearing_position
        p4168582468: Chiller_1.Thrust_bearing_position
    Label (857,788 135x30), "Liquid valve position"
    Textfield (878,814 92x25), "%1.0f %%", text variable: Chiller_1.Feedback_liquid_valve
        p4168582468: Chiller_1.Feedback_liquid_valve
    Textfield (780,753 78x25), "%1.2f bar", text variable: Chiller_1.Oil_Filter_Drop
        p4168582468: Chiller_1.Oil_Filter_Drop
    Label (778,732 83x22), "Oil filter drop"
    Textfield (667,814 92x25), "%1.0f %%", text variable: Chiller_1.Liquid_valve_output
        p4168582468: Chiller_1.Liquid_valve_output
    Label (646,788 135x30), "Liquid valve order"
    Textfield (780,703 78x25), "%1.2f bar", text variable: Chiller_1.Press_oil_receiver
        p4168582468: Chiller_1.Press_oil_receiver
    Label (752,682 135x22), "Oil pressure receiver"
    Textfield (780,654 78x25), "%1.1f °C", text variable: Chiller_1.Oil_temp_receiver
        p4168582468: Chiller_1.Oil_temp_receiver
    Label (748,633 143x22), "Oil temperature receiver"
    Textfield (780,605 78x25), "%1.2f bar", text variable: Chiller_1.Oil_diff_pressure
        p4168582468: Chiller_1.Oil_diff_pressure
    Label (769,584 101x22), "Oil diff pressure"
    Label (738,136 105x24), "Prerotary position"
    Textfield (754,159 72x25), "%1.0f %%", text variable: Chiller_1.Feedback_PRV
        p4168582468: Chiller_1.Feedback_PRV
    Label (746,83 87x24), "VGD position"
    Textfield (753,106 72x25), "%1.0f %%", text variable: Chiller_1.Feedback_VGD
        p4168582468: Chiller_1.Feedback_VGD
    Label (746,31 87x24), "Stall detector"
    Textfield (753,54 72x25), "%1.2f V", text variable: Chiller_1.Stall_detector
        p4168582468: Chiller_1.Stall_detector
    Label (1067,211 171x24), "Suction pressure saturated"
    Textfield (1116,234 72x25), "%1.1f °C", text variable: Chiller_1.Suction_saturated_temp
        p4168582468: Chiller_1.Suction_saturated_temp
    Textfield (1116,291 72x25), "%1.1f bara", text variable: Chiller_1.Press_suction_compr
        p4168582468: Chiller_1.Press_suction_compr
    Label (1067,268 171x24), "Suction pressure"
    Textfield (1116,368 72x25), "%1.1f °C", text variable: Chiller_1.Theta_out
        p4168582468: Chiller_1.Theta_out
    Label (1111,345 83x24), "Theta out"
    Label (1196,557 84x27), "CW pressure"
    Textfield (1200,581 77x25), "%1.2f bar", text variable: Chiller_1.Press_chilled_medium_out
        p4168582468: Chiller_1.Press_chilled_medium_out
    Textfield (1200,710 77x25), "%1.2f bar", text variable: Chiller_1.Press_chilled_medium_in
        p4168582468: Chiller_1.Press_chilled_medium_in
    Label (1196,686 84x27), "CW pressure"
    Textfield (1170,506 72x25), "%1.1f °C", text variable: Chiller_1.Temp_chilled_medium_out
        p4168582468: Chiller_1.Temp_chilled_medium_out
    Label (1146,483 121x24), "Chilled water outlet"
    Label (1146,428 121x24), "CW setpoint"
    Textfield (1170,451 72x25), "%1.1f °C", text variable: Chiller_1.SP_CW_controller
        p4168582468: Chiller_1.SP_CW_controller
    Label (1252,619 84x30), "Diff pressure"
    Textfield (1256,648 77x25), "%1.2f bar", text variable: Chiller_1.dP_CW
        p4168582468: Chiller_1.dP_CW
    Textfield (1170,783 72x25), "%1.1f °C", text variable: Chiller_1.Temp_chilled_medium_in
        p4168582468: Chiller_1.Temp_chilled_medium_in
    Label (1146,760 121x24), "Chilled water inlet"
    Group (6,271 190x25)
        Rectangle (0,0 190x25)
        Label (0,2 105x21), "Running"
        Lamp1 (166,3 23x20), variable: Chiller_1.Unit_running, style: Lamp-Lamp1-Green
    Group (6,163 190x25)
        Rectangle (0,0 190x25)
        Label (1,2 105x21), "Auto"
        Lamp1 (166,3 23x20), variable: Chiller_1.Unit_auto, style: Lamp-Lamp1-Green
    Group (6,199 190x25)
        Rectangle (0,0 190x25)
        Label (0,2 105x21), "Remote"
        Lamp1 (166,3 23x20), variable: Chiller_1.Unit_remote, style: Lamp-Lamp1-Green
    Group (6,235 190x25)
        Rectangle (0,0 190x25)
        Label (0,2 105x21), "Manual"
        Lamp1 (166,3 23x20), variable: Chiller_1.Unit_manual, style: Lamp-Lamp1-Green
    Group (6,307 190x25)
        Rectangle (0,0 190x25)
        Label (1,2 105x21), "Available"
        Lamp1 (166,3 23x20), variable: Chiller_1.Unit_available, style: Lamp-Lamp1-Green
    Group (6,343 190x25)
        Rectangle (0,0 190x25)
        Label (0,2 130x21), "Start switch"
        Lamp1 (166,3 23x20), variable: Chiller_1.Unit_start_switch, style: Lamp-Lamp1-Green
    Group (6,381 190x25)
        Rectangle (0,0 190x25)
        Label (0,2 160x21), "Comms sequence"
        Lamp1 (166,3 23x20), variable: not.Sequence.A_Comms_chiller_1, style: Lamp-Lamp1-Green
    Label (912,265 95x24), "Oil temp comp."
    Textfield (923,288 72x25), "%1.1f °C", text variable: Chiller_1.Temp_oil_inlet_compr
        p4168582468: Chiller_1.Temp_oil_inlet_compr
    Label (902,324 115x24), "Oil pressure [HP]"
    Textfield (923,347 72x25), "%1.2f bar", text variable: Chiller_1.Press_oil_compr
        p4168582468: Chiller_1.Press_oil_compr
    Image (921,41 317x130), invisible if: Chiller_1.Unit_alarm, image: ImagePool.ALARM
    Image (921,41 317x130), invisible if: Chiller_1.Unit_trip, image: ImagePool.TRIP
    Label (7,87 89x30), "Mode"
    Label (106,87 89x30), "Status"
    Rectangle (334,160 48x246)
    Image (238,160 48x246), image: ImagePool.CapBarTranparant
    BarDisplayImage (239,161 46x242), value: Sequence.Seq_cap_order_C1, style: BarDisplayImage-Gray, scale format: %.0f, scale 0..100
        p3451962224: ImagePool.Invisible
    Rectangle (673,210 36x36), colour toggle: Chiller_1.Unit_running
    Rectangle (673,210 36x36), colour toggle: Chiller_1.Unit_alarm
    Rectangle (673,210 36x36), colour toggle: Chiller_1.Unit_trip
    Image (334,160 48x246), image: ImagePool.CapBarTranparant
    BarDisplayImage (335,161 46x242), value: Chiller_1.Chiller_capacity_t1, style: BarDisplayImage-Gray, scale format: %.0f, scale 0..100
        p3451962224: ImagePool.Invisible
    Rectangle (493,624 28x52)
    Image (493,624 29x54), image: ImagePool.CapBarTranparant
    BarDisplayImage (494,625 27x51), value: Chiller_1.Liquid_level_condenser, style: BarDisplayImage-Gray, scale format: %.0f, scale 0..100
        p3451962224: ImagePool.Invisible
    Image (95,742 147x16), image: ImagePool.PipeGreen_1_Horizontal
    Textfield (605,753 92x25), "%1.1f °C", text variable: Chiller_1.Liquid_line_temp
        p4168582468: Chiller_1.Liquid_line_temp
    Label (595,727 113x30), "Liquid line temp"
    Label (435,287 154x30), "Vibration comp motor"
    Textfield (474,344 77x25), "%1.1f mm/s", text variable: Chiller_1.Vibration_compressor_NDE
        p4168582468: Chiller_1.Vibration_compressor_NDE
    Textfield (474,314 77x25), "%1.1f mm/s", text variable: Chiller_1.Vibration_compressor_DE
        p4168582468: Chiller_1.Vibration_compressor_DE
    Label (429,314 37x25), "DE"
    Label (429,344 37x25), "NDE"
    Image (228,490 57x88), image: ImagePool.Valve_3
    Label (115,461 105x30), "Sea water valve order"
    Textfield (129,492 76x25), "%1.0f %%", text variable: Chiller_1.Control_signal_SW_valve
        p4168582468: Chiller_1.Control_signal_SW_valve
    Label (281,461 105x30), "Sea water valve pos"
    Textfield (295,492 76x25), "%1.0f %%", text variable: Chiller_1.Feedback_sea_water_valve
        p4168582468: Chiller_1.Feedback_sea_water_valve
    Group (37,610 180x72)
        Rectangle (0,0 180x72)
        Label (0,0 180x72), "Sea water valve Pos. 100% = Max. overboard Pos. 0% = Max. recirculation"
    Label (521,115 83x22), "Motor speed"
    Textfield (526,136 72x25), "%1.0f Hz", text variable: Chiller_1.Opt_speed_VFD_Hz
        p4168582468: Chiller_1.Opt_speed_VFD_Hz
END_VISUALIZATION

// /Chiller_1_Oil
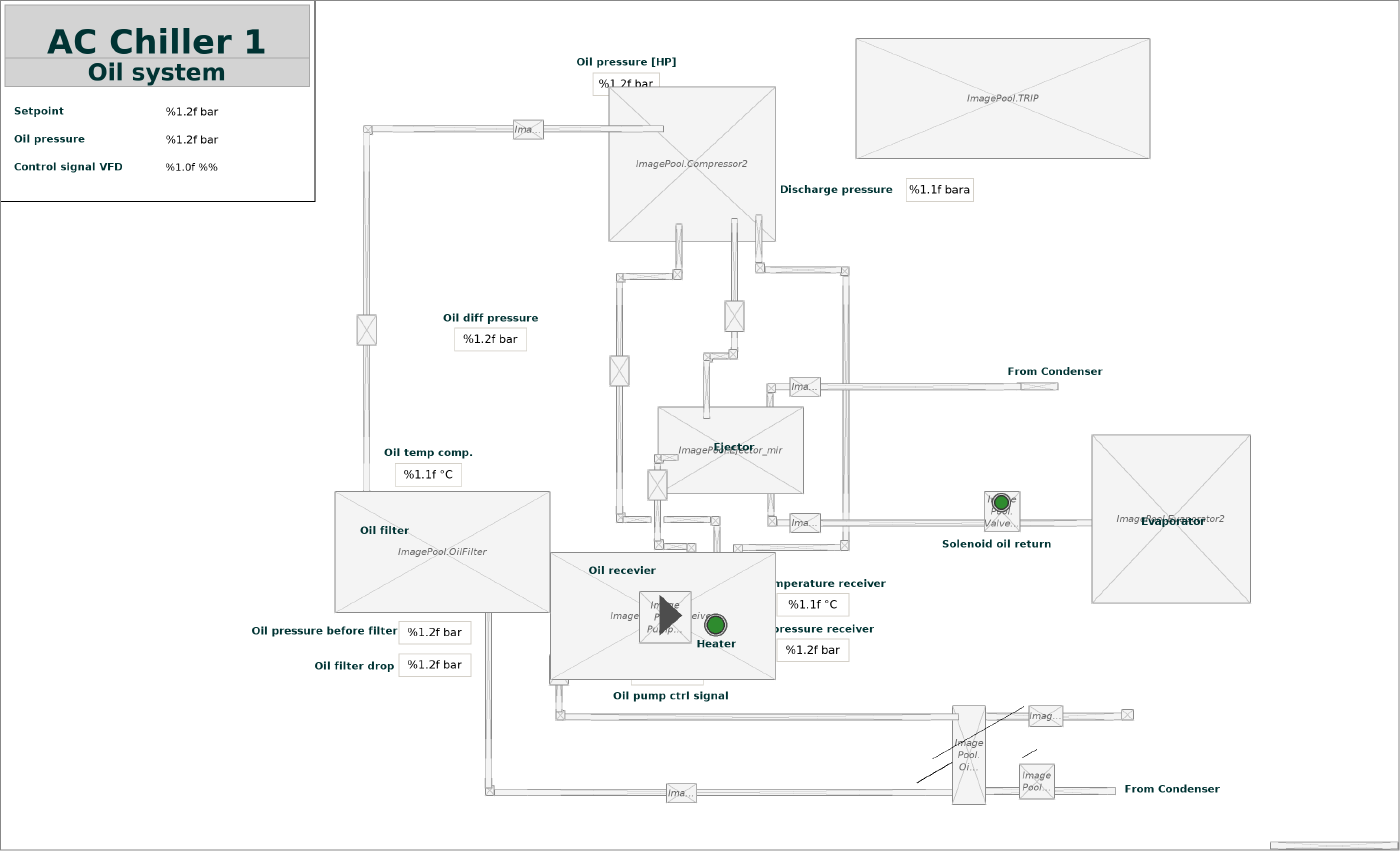
VISUALIZATION Chiller_1_Oil  // 1507x917
    Image (1094,412 45x8), angle 180, image: ImagePool.PipeBlack_1S_H_Faded
    Rectangle (0,0 339x217)
    Image (1367,907 138x8), angle 270, image: ImagePool.PipeGrey_1S_Horizontal
    Image (1053,768 155x8), image: ImagePool.PipeGrey_1S_Horizontal
    Image (1207,764 13x12), image: ImagePool.PipeGrey_3_LU
    Textfield (5,5 328x80), "AC Chiller 1"
    Label (1093,387 97x27), "From Condenser"
    Label (835,191 129x27), "Discharge pressure"
    Textfield (975,192 73x25), "%1.1f bara", text variable: Chiller_1.Press_discharge_compr
        p4168582468: Chiller_1.Press_discharge_compr
    Label (1029,573 106x27), "Solenoid oil return"
    Textfield (429,704 78x25), "%1.2f bar", text variable: Chiller_1.Oil_Filter_Drop
        p4168582468: Chiller_1.Oil_Filter_Drop
    Label (340,707 83x22), "Oil filter drop"
    Textfield (836,688 78x25), "%1.2f bar", text variable: Chiller_1.Press_oil_receiver
        p4168582468: Chiller_1.Press_oil_receiver
    Label (808,667 135x22), "Oil pressure receiver"
    Textfield (836,639 78x25), "%1.1f °C", text variable: Chiller_1.Oil_temp_receiver
        p4168582468: Chiller_1.Oil_temp_receiver
    Label (804,618 143x22), "Oil temperature receiver"
    Textfield (489,353 78x25), "%1.2f bar", text variable: Chiller_1.Oil_diff_pressure
        p4168582468: Chiller_1.Oil_diff_pressure
    Label (478,332 101x22), "Oil diff pressure"
    Label (414,476 95x24), "Oil temp comp."
    Textfield (425,499 72x25), "%1.1f °C", text variable: Chiller_1.Temp_oil_inlet_compr
        p4168582468: Chiller_1.Temp_oil_inlet_compr
    Label (617,55 115x24), "Oil pressure [HP]"
    Textfield (638,78 72x25), "%1.2f bar", text variable: Chiller_1.Press_oil_compr
        p4168582468: Chiller_1.Press_oil_compr
    Image (921,41 317x130), invisible if: not.Chiller_1.Unit_alarm, image: ImagePool.ALARM
    Image (921,41 317x130), invisible if: not.Chiller_1.Unit_trip, image: ImagePool.TRIP
    Textfield (5,62 328x31), "Oil system"
    Textfield (178,109 57x23), "%1.2f bar", tooltip "Chiller_1.SP_oil_pressure_diff", text variable: Chiller_1.SP_oil_pressure_diff
    Label (12,105 106x30), "Setpoint"
    Textfield (178,139 57x23), "%1.2f bar", tooltip "Chiller_1.Oil_diff_pressure", text variable: Chiller_1.Oil_diff_pressure
    Label (12,135 107x30), "Oil pressure"
    Textfield (178,169 57x23), "%1.0f %%", tooltip "Chiller_1.SP_freq_oil_pump_VFD", text variable: Chiller_1.SP_freq_oil_pump_VFD
    Label (12,165 109x30), "Control signal VFD"
    Textfield (679,713 78x25), "%1.2f Hz", tooltip "Chiller_1.SP_freq_oil_pump_VFD", text variable: Chiller_1.Press_oil_receiver
    Label (655,739 135x22), "Oil pump ctrl signal"
    Textfield (429,669 78x25), "%1.2f bar", text variable: Chiller_1.Oil_pressure_before_filter
        p4168582468: Chiller_1.Oil_pressure_before_filter
    Label (276,669 147x22), "Oil pressure before filter"
    Label (1210,837 106x27), "From Condenser"
    Image (655,93 180x167), image: ImagePool.Compressor2
    Image (1051,848 150x8), angle 180, image: ImagePool.PipeBlack_1S_H_Faded
    Image (798,586 108x7), image: ImagePool.PipeBlack_1_Horizontal
    Image (907,297 7x286), image: ImagePool.PipeBlack_1_Vertical
    Image (391,135 10x10), image: ImagePool.PipeBlack_1_RD
    Image (522,846 10x11), image: ImagePool.PipeBlack_1_RU
    Image (1107,760 37x23), image: ImagePool.Arrow gray right
    Image (836,560 348x7), image: ImagePool.PipeBlack_1_Horizontal
    Image (1175,468 171x182), image: ImagePool.Evaporator2
    Image (826,512 7x44), image: ImagePool.PipeBlack_1_Vertical
    Image (826,556 10x11), image: ImagePool.PipeBlack_1_RU
    Image (789,596 7x28), image: ImagePool.PipeBlack_1_Vertical
    Image (789,586 10x10), image: ImagePool.PipeBlack_1_RD
    Image (904,582 10x11), image: ImagePool.PipeBlack_1_LU
    Image (850,553 33x21), image: ImagePool.Arrow black left
    Image (904,287 10x10), image: ImagePool.PipeBlack_1_LD
    Image (823,287 83x7), image: ImagePool.PipeBlack_1_Horizontal
    Image (813,283 10x11), image: ImagePool.PipeBlack_1_RU
    Image (813,231 7x52), image: ImagePool.PipeBlack_1_Vertical
    Image (825,413 10x10), image: ImagePool.PipeBlack_1_RD
    Image (834,413 265x7), image: ImagePool.PipeBlack_1_Horizontal
    Image (825,423 7x28), image: ImagePool.PipeBlack_1_Vertical
    Image (708,438 157x94), image: ImagePool.Ejector_mir
    Image (850,406 33x21), image: ImagePool.Arrow black left
    Image (532,850 500x7), image: ImagePool.PipeBlack_1_Horizontal
    Image (1025,760 36x107), image: ImagePool.OilHeatExchanger
    Image (605,769 427x7), image: ImagePool.PipeBlack_1_Horizontal
    Image (598,765 10x11), image: ImagePool.PipeBlack_1_RU
    Image (598,670 7x97), image: ImagePool.PipeBlack_1_Vertical
    Image (598,660 10x10), image: ImagePool.PipeBlack_1_RD
    Image (605,660 19x7), image: ImagePool.PipeBlack_1_Horizontal
    Image (591,705 21x33), image: ImagePool.Arrow black down
    Image (717,844 33x21), image: ImagePool.Arrow black left
    Image (768,566 7x50), image: ImagePool.PipeBlack_1_Vertical
    Image (765,556 10x10), image: ImagePool.PipeBlack_1_LD
    Image (714,556 51x7), image: ImagePool.PipeBlack_1_Horizontal
    Image (704,581 10x11), image: ImagePool.PipeBlack_1_RU
    Image (704,499 7x84), image: ImagePool.PipeBlack_1_Vertical
    Image (704,489 10x10), image: ImagePool.PipeBlack_1_RD
    Image (711,489 19x7), image: ImagePool.PipeBlack_1_Horizontal
    Image (697,506 21x33), image: ImagePool.Arrow black down
    Image (714,585 28x7), image: ImagePool.PipeBlack_1_Horizontal
    Image (739,585 10x10), image: ImagePool.PipeBlack_1_LD
    Image (742,595 7x21), image: ImagePool.PipeBlack_1_Vertical
    Image (592,595 243x137), image: ImagePool.OilReceiver
    Image (400,135 314x7), image: ImagePool.PipeBlack_1_Horizontal
    Label (630,604 80x22), "Oil recevier"
    Image (522,553 7x296), image: ImagePool.PipeBlack_1_Vertical
    Image (519,544 10x10), image: ImagePool.PipeBlack_1_LD
    Image (400,544 120x7), image: ImagePool.PipeBlack_1_Horizontal
    Image (391,540 10x11), image: ImagePool.PipeBlack_1_RU
    Image (391,142 7x400), image: ImagePool.PipeBlack_1_Vertical
    Image (663,552 10x11), image: ImagePool.PipeBlack_1_RU
    Image (663,301 7x253), image: ImagePool.PipeBlack_1_Vertical
    Image (663,294 10x10), image: ImagePool.PipeBlack_1_RD
    Image (670,294 54x7), image: ImagePool.PipeBlack_1_Horizontal
    Image (656,383 21x33), image: ImagePool.Arrow black down
    Image (670,556 31x7), image: ImagePool.PipeBlack_1_Horizontal
    Image (727,241 7x53), image: ImagePool.PipeBlack_1_Vertical
    Image (724,290 10x11), image: ImagePool.PipeBlack_1_LU
    Image (757,380 10x10), image: ImagePool.PipeBlack_1_RD
    Image (764,380 22x7), image: ImagePool.PipeBlack_1_Horizontal
    Image (787,235 7x144), image: ImagePool.PipeBlack_1_Vertical
    Image (784,376 10x11), image: ImagePool.PipeBlack_1_LU
    Image (757,388 7x63), image: ImagePool.PipeBlack_1_Vertical
    Image (780,324 21x33), image: ImagePool.Arrow black down
    Label (750,471 80x22), "Ejector"
    Label (1223,551 80x22), "Evaporator"
    Image (384,339 21x33), image: ImagePool.Arrow black up
    Image (552,129 33x21), image: ImagePool.Arrow black right
    Image (360,529 232x131), image: ImagePool.OilFilter
    Label (387,561 54x22), "Oil filter"
    Line (987,843) (1025,821)
    Line (1100,816) (1116,807)
    Line (1004,817) (1102,761)
    Image (1097,823 38x38), image: ImagePool.RegValve
    Image (688,637 56x56), image: ImagePool.Pump_Large_3
    Polygon (710,660) (710,641) (734,663) (710,684) (710,676), colour toggle: Chiller_1.Comp_oil_pump
    Lamp1 (756,656 29x35), variable: Chiller_1.Oil_heater, style: Lamp-Lamp1-Green
    Label (744,683 55x22), "Heater"
    Image (1059,529 39x44), image: ImagePool.Valve_2
    Lamp1 (1066,529 24x25), variable: Chiller_1.Solenoid_oil_return, style: Lamp-Lamp1-Green
END_VISUALIZATION

